CR140_Horz_Cyl_3(
	Auto:=OP140_AutoSelected , 
	Manual:=OP140_ManualSelected , 
	ErrorActive:=OP140_ErrorActive , 
	ResetPB:=OP140_HMI_Reset , 
	Sensor1:=I140_HORZ_SUP3_CYL_REVI1310_6  , 
	Sensor2:=I140_HORZ_SUP3_CYL_FWDI1310_7  , 
	ManualPB1:= , 
	ManualPB2:= , 
	AutoCmd1:= , 
	AutoCmd2:= , 
	OperationEnable:=OperationEnable , 
	SafeHome:= , 
	SafeWork:= , 
	HomingCmd1:= , 
	Pulse_1Sec:=Pulse_Block.Q1Hz , 
	BlinkingBit:= , 
	TimeOut1:=10 , 
	TimeOut2:=10 , 
	TimeOut3:=10 , 
	Solenoid1=>O140_HORZ_SUP3_CYL_REV_Q1343_0 , 
	Solenoid2=>O140_HORZ_SUP3_CYL_FWD_Q1343_1  , 
	AlarmSensor1=>berror[1331] , 
	AlarmSensor2=>berror[1332] , 
	AlarmSolenoid1=>berror[1333] , 
	AlarmSolenoid2=>berror[1334] , 
	AllSignal=>berror[1335] , 
	AlarmPresent=> , 
	Position1=> , 
	Position2=> , 
	HomeSensorBlink=> , 
	WorkSensorBlink=> , 
	Status:=OP140_GVL.CR140_Horz_Cyl_1_Status );
	
	
	//Vertical Cylinder 1
OP140_Gvl.CR140_Vert_Cyl_1_Status:=0;
// Safe Home
IF (SR140_HMI_Vert_Servo_MC1.actualPosition<=50) THEN 
	CR140_Vert_Cyl_1.SafeHome:= TRUE;
	ELSE
		CR140_Vert_Cyl_1.SafeHome:= FALSE;
	END_IF
	//Safe Work
IF(TRUE) THEN 
CR140_Vert_Cyl_1.SafeWork:=TRUE;
ELSE
	CR140_Vert_Cyl_1.SafeWork:=FALSE;
	END_IF
//Manual PB 1
IF(OP140_HMI_Vert_Cyl1_Home_PB) THEN
	CR140_Vert_Cyl_1.ManualPB1:=TRUE;
	ELSE
		CR140_Vert_Cyl_1.ManualPB1:=FALSE;
	END_IF
//Manual PB2 
IF(OP140_HMI_Vert_Cyl1_Work_PB) THEN
	CR140_Vert_Cyl_1.ManualPB2:=TRUE;
	ELSE
		CR140_Vert_Cyl_1.ManualPB2:=FALSE;
	END_IF	

	

CR140_Vert_Cyl_1(
	Auto:=OP140_AutoSelected , 
	Manual:=OP140_ManualSelected , 
	ErrorActive:=OP140_ErrorActive , 
	ResetPB:=OP140_HMI_Reset , 
	Sensor1:=I140_VERT_SUP1_CYL_REVI1301_2  , 
	Sensor2:=I140_VERT_SUP1_CYL_FWDI1301_3  , 
	ManualPB1:= , 
	ManualPB2:= , 
	AutoCmd1:= , 
	AutoCmd2:= , 
	OperationEnable:=OperationEnable , 
	SafeHome:= , 
	SafeWork:= , 
	HomingCmd1:= , 
	Pulse_1Sec:=Pulse_Block.Q1Hz  , 
	BlinkingBit:= , 
	TimeOut1:=10 , 
	TimeOut2:=10 , 
	TimeOut3:=10 , 
	Solenoid1=>O140_VERT_SUP1_CYL_REV_Q1341_2  , 
	Solenoid2=>O140_VERT_SUP1_CYL_FWD_Q1341_3 , 
	AlarmSensor1=> berror[1306], 
	AlarmSensor2=>berror[1307] , 
	AlarmSolenoid1=>berror[1308] , 
	AlarmSolenoid2=>berror[1309] , 
	AllSignal=>berror[1310],
	AlarmPresent=> , 
	Position1=> , 
	Position2=> , 
	HomeSensorBlink=> , 
	WorkSensorBlink=> , 
	Status:=OP140_Gvl.CR140_Vert_Cyl_1_Status );
	
		//Vertical Cylinder 2
CR140_Vert_Cyl_2_Status:=0;
// Safe Home
IF (SR140_HMI_Vert_Servo_MC2.actualPosition<=50) THEN 
	CR140_Vert_Cyl_2.SafeHome:= TRUE;
	ELSE
		CR140_Vert_Cyl_2.SafeHome:= FALSE;
	END_IF
	//Safe Work
IF(TRUE) THEN 
CR140_Vert_Cyl_2.SafeWork:=TRUE;
ELSE
	CR140_Vert_Cyl_2.SafeWork:=FALSE;
	END_IF
//Manual PB 1
IF(OP140_HMI_Vert_Cyl2_Home_PB) THEN
	CR140_Vert_Cyl_2.ManualPB1:=TRUE;
	ELSE
		CR140_Vert_Cyl_2.ManualPB1:=FALSE;
	END_IF
//Manual PB2 
IF(OP140_HMI_Vert_Cyl2_Work_PB) THEN
	CR140_Vert_Cyl_2.ManualPB2:=TRUE;
	ELSE
		CR140_Vert_Cyl_2.ManualPB2:=FALSE;
	END_IF	

	

CR140_Vert_Cyl_2(
	Auto:=OP140_AutoSelected , 
	Manual:=OP140_ManualSelected , 
	ErrorActive:=OP140_ErrorActive , 
	ResetPB:=OP140_HMI_Reset , 
	Sensor1:=I140_VERT_SUP2_CYL_REVI1310_2 , 
	Sensor2:=I140_VERT_SUP2_CYL_FWDI1310_3 , 
	ManualPB1:= , 
	ManualPB2:= , 
	AutoCmd1:= , 
	AutoCmd2:= , 
	OperationEnable:=OperationEnable , 
	SafeHome:= , 
	SafeWork:= , 
	HomingCmd1:= , 
	Pulse_1Sec:=Pulse_Block.Q1Hz , 
	BlinkingBit:= , 
	TimeOut1:=10 , 
	TimeOut2:=10 , 
	TimeOut3:=10 , 
	Solenoid1=>O140_VERT_SUP2_CYL_REV_Q1342_2 , 
	Solenoid2=>O140_VERT_SUP2_CYL_FWD_Q1342_3  , 
	AlarmSensor1=>berror[1321] , 
	AlarmSensor2=>berror[1322] , 
	AlarmSolenoid1=>berror[1323] , 
	AlarmSolenoid2=>berror[1324] , 
	AllSignal=>berror[1325] , 
	AlarmPresent=> , 
	Position1=> , 
	Position2=> , 
	HomeSensorBlink=> , 
	WorkSensorBlink=> , 
	Status:=CR140_Vert_Cyl_2_Status );
	
		//Vertical Cylinder 3
CR140_Vert_Cyl_3_Status:=0;
// Safe Home
IF (SR140_HMI_Vert_Servo_MC3.actualPosition<=50) THEN 
	CR140_Vert_Cyl_3.SafeHome:= TRUE;
	ELSE
		CR140_Vert_Cyl_3.SafeHome:= FALSE;
	END_IF
	//Safe Work
IF(TRUE) THEN 
   CR140_Vert_Cyl_3.SafeWork:=TRUE;
ELSE
	CR140_Vert_Cyl_3.SafeWork:=FALSE;
END_IF
//Manual PB 1
IF(OP140_HMI_Vert_Cyl3_Home_PB) THEN
	CR140_Vert_Cyl_3.ManualPB1:=TRUE;
	ELSE
		CR140_Vert_Cyl_3.ManualPB1:=FALSE;
	END_IF
//Manual PB2 
IF(OP140_HMI_Vert_Cyl3_Work_PB) THEN
	CR140_Vert_Cyl_3.ManualPB2:=TRUE;
	ELSE
		CR140_Vert_Cyl_3.ManualPB2:=FALSE;
	END_IF	

	

CR140_Vert_Cyl_3(
	Auto:=OP140_AutoSelected , 
	Manual:=OP140_ManualSelected , 
	ErrorActive:=OP140_ErrorActive , 
	ResetPB:=OP140_HMI_Reset , 
	Sensor1:=I140_VERT_SUP3_CYL_REVI1311_0 , 
	Sensor2:=I140_VERT_SUP3_CYL_FWDI1311_1  , 
	ManualPB1:= , 
	ManualPB2:= , 
	AutoCmd1:= , 
	AutoCmd2:= , 
	OperationEnable:= OperationEnable, 
	SafeHome:= , 
	SafeWork:= , 
	HomingCmd1:= , 
	Pulse_1Sec:=Pulse_Block.Q1Hz , 
	BlinkingBit:= , 
	TimeOut1:=10 , 
	TimeOut2:=10 , 
	TimeOut3:=10 , 
	Solenoid1=>O140_VERT_SUP3_CYL_REV_Q1343_2 , 
	Solenoid2=>O140_VERT_SUP3_CYL_FWD_Q1343_3  , 
	AlarmSensor1=>berror[1336] , 
	AlarmSensor2=>berror[1337] , 
	AlarmSolenoid1=>berror[1338] , 
	AlarmSolenoid2=>berror[1339] , 
	AllSignal=>berror[1340] , 
	AlarmPresent=> , 
	Position1=> , 
	Position2=> , 
	HomeSensorBlink=> , 
	WorkSensorBlink=> , 
	Status:=CR140_Vert_Cyl_3_Status );
	
		//Top Wipe Cylinder 
CR140_Wipe_Cyl_1_Status:=0;
// Safe Home
IF (TRUE) THEN 
	CR140_Top_Wipe_Cyl_1.SafeHome:= TRUE;
	ELSE
		CR140_Top_Wipe_Cyl_1.SafeHome:= FALSE;
	END_IF
	//Safe Work
IF(SR140_Vert_Servo_Ctrl_1.Axis_In_Home) THEN 
CR140_Top_Wipe_Cyl_1.SafeWork:=TRUE;
ELSE
	CR140_Top_Wipe_Cyl_1.SafeWork:=FALSE;
	END_IF
//Manual PB 1
IF(OP140_HMI_Wipe_Cyl1_Home_PB) THEN
	CR140_Top_Wipe_Cyl_1.ManualPB1:=TRUE;
	ELSE
		CR140_Top_Wipe_Cyl_1.ManualPB1:=FALSE;
	END_IF
//Manual PB2 
IF(OP140_HMI_Wipe_Cyl1_Work_PB) THEN
	CR140_Top_Wipe_Cyl_1.ManualPB2:=TRUE;
	ELSE
		CR140_Top_Wipe_Cyl_1.ManualPB2:=FALSE;
	END_IF	

	

CR140_Top_Wipe_Cyl_1(
	Auto:=OP140_AutoSelected , 
	Manual:=OP140_ManualSelected, 
	ErrorActive:=OP140_ErrorActive , 
	ResetPB:=OP140_HMI_Reset , 
	Sensor1:=I140_WIPE1_CYL_REVI1301_4, 
	Sensor2:=I140_WIPE1_CYL_FWDI1301_5 , 
	ManualPB1:= , 
	ManualPB2:= , 
	AutoCmd1:= , 
	AutoCmd2:= , 
	OperationEnable:=OperationEnable , 
	SafeHome:= , 
	SafeWork:= , 
	HomingCmd1:= , 
	Pulse_1Sec:=Pulse_Block.Q1Hz , 
	BlinkingBit:= , 
	TimeOut1:=10 , 
	TimeOut2:=10 , 
	TimeOut3:=10 , 
	Solenoid1=>O140_WIPE1_CYL_REV_Q1341_6 , 
	Solenoid2=>O140_WIPE1_CYL_FWD_Q1341_7  , 
	AlarmSensor1=>berror[1311] , 
	AlarmSensor2=>berror[1312] , 
	AlarmSolenoid1=>berror[1313] , 
	AlarmSolenoid2=>berror[1314] , 
	AllSignal=>berror[1315] , 
	AlarmPresent=> , 
	Position1=> , 
	Position2=> , 
	HomeSensorBlink=> , 
	WorkSensorBlink=> , 
	Status:=CR140_Wipe_Cyl_1_Status );
	
	//Top Wipe Cyl 2
	CR140_Wipe_Cyl_2_Status:=0;
// Safe Home
IF (TRUE) THEN 
	CR140_Top_Wipe_Cyl_2.SafeHome:= TRUE;
	ELSE
		CR140_Top_Wipe_Cyl_2.SafeHome:= FALSE;
	END_IF
	//Safe Work
IF(SR140_Vert_Servo_Ctrl_2.Axis_In_Home) THEN 
CR140_Top_Wipe_Cyl_2.SafeWork:=TRUE;
ELSE
	CR140_Top_Wipe_Cyl_2.SafeWork:=FALSE;
	END_IF
//Manual PB 1
IF(OP140_HMI_Wipe_Cyl2_Home_PB) THEN
	CR140_Top_Wipe_Cyl_2.ManualPB1:=TRUE;
	ELSE
		CR140_Top_Wipe_Cyl_2.ManualPB1:=FALSE;
	END_IF
//Manual PB2 
IF(OP140_HMI_Wipe_Cyl2_Work_PB) THEN
	CR140_Top_Wipe_Cyl_2.ManualPB2:=TRUE;
	ELSE
		CR140_Top_Wipe_Cyl_2.ManualPB2:=FALSE;
	END_IF	

	

CR140_Top_Wipe_Cyl_2(
	Auto:=OP140_AutoSelected , 
	Manual:=OP140_ManualSelected , 
	ErrorActive:=OP140_ErrorActive , 
	ResetPB:=OP140_HMI_Reset , 
	Sensor1:=I140_WIPE2_CYL_REVI1310_4 , 
	Sensor2:=I140_WIPE2_CYL_FWDI1310_5  , 
	ManualPB1:= , 
	ManualPB2:= , 
	AutoCmd1:= , 
	AutoCmd2:= , 
	OperationEnable:=OperationEnable , 
	SafeHome:= , 
	SafeWork:= , 
	HomingCmd1:= , 
	Pulse_1Sec:=Pulse_Block.Q1Hz , 
	BlinkingBit:= , 
	TimeOut1:=10 , 
	TimeOut2:=10 , 
	TimeOut3:=10 , 
	Solenoid1=>O140_WIPE2_CYL_REV_Q1342_6  , 
	Solenoid2=>O140_WIPE2_CYL_FWD_Q1342_7 , 
	AlarmSensor1=>berror[1326] , 
	AlarmSensor2=>berror[1327] , 
	AlarmSolenoid1=>berror[1328] , 
	AlarmSolenoid2=>berror[1329] , 
	AllSignal=>berror[1330] , 
	AlarmPresent=> , 
	Position1=> , 
	Position2=> , 
	HomeSensorBlink=> , 
	WorkSensorBlink=> , 
	Status:=CR140_Wipe_Cyl_2_Status );
	
//Wipe Cylinder 3

CR140_Wipe_Cyl_3_Status:=0;
// Safe Home
IF (TRUE) THEN 
	CR140_Top_Wipe_Cyl_3.SafeHome:= TRUE;
	ELSE
		CR140_Top_Wipe_Cyl_3.SafeHome:= FALSE;
	END_IF
	//Safe Work
IF(SR140_Vert_Servo_Ctrl_3.Axis_In_Home) THEN 
CR140_Top_Wipe_Cyl_3.SafeWork:=TRUE;
ELSE
	CR140_Top_Wipe_Cyl_3.SafeWork:=FALSE;
	END_IF
//Manual PB 1
IF(OP140_HMI_Wipe_Cyl3_Home_PB) THEN
	CR140_Top_Wipe_Cyl_3.ManualPB1:=TRUE;
	ELSE
		CR140_Top_Wipe_Cyl_3.ManualPB1:=FALSE;
	END_IF
//Manual PB2 
IF(OP140_HMI_Wipe_Cyl3_Work_PB) THEN
	CR140_Top_Wipe_Cyl_3.ManualPB2:=TRUE;
	ELSE
		CR140_Top_Wipe_Cyl_3.ManualPB2:=FALSE;
	END_IF	

	

CR140_Top_Wipe_Cyl_3(
	Auto:=OP140_AutoSelected , 
	Manual:=OP140_ManualSelected , 
	ErrorActive:=OP140_ErrorActive , 
	ResetPB:=OP140_HMI_Reset , 
	Sensor1:=I140_WIPE3_CYL_REVI1311_2 , 
	Sensor2:=I140_WIPE3_CYL_FWDI1311_3  , 
	ManualPB1:= , 
	ManualPB2:= , 
	AutoCmd1:= , 
	AutoCmd2:= , 
	OperationEnable:=OperationEnable , 
	SafeHome:= , 
	SafeWork:= , 
	HomingCmd1:= , 
	Pulse_1Sec:= Pulse_Block.Q1Hz, 
	BlinkingBit:= , 
	TimeOut1:=10 , 
	TimeOut2:=10 , 
	TimeOut3:= 10, 
	Solenoid1=>O140_WIPE3_CYL_REV_Q1343_6 , 
	Solenoid2=>O140_WIPE3_CYL_FWD_Q1343_7  , 
	AlarmSensor1=>berror[1341] , 
	AlarmSensor2=>berror[1342] , 
	AlarmSolenoid1=>berror[1343] , 
	AlarmSolenoid2=>berror[1344] , 
	AllSignal=>berror[1345] , 
	AlarmPresent=> , 
	Position1=> , 
	Position2=> , 
	HomeSensorBlink=> , 
	WorkSensorBlink=> , 
	Status:=CR140_Wipe_Cyl_3_Status );
		
	
	//Vertical Servo 1
	
	// Safe to Move
	
	IF CR140_Top_Wipe_Cyl_1.Position1	AND CR140_Horz_Cyl_1.Sensor2  AND CR140_Vert_Cyl_1.Position2 THEN //OR SR140_HMI_Vert_Servo_MC1.actualPosition <=50)	THEN
		
		OP140_Servo1_Safety:=TRUE;
		ELSE
			OP140_Servo1_Safety:=FALSE;
		END_IF

		//LH Vertical Servo 1
SR140_Vert_Servo_1(
	bAxis1_Ref_Switch:= , 
	bInit:= , 
	bErrorReset:=OP140_HMI_Reset OR Servo_Reset, 
	bEnable:= Servo_Enable, 
	bMoveVelocity:= , 
	bHalt:= , 
	bManualMode:=OP140_ManualSelected , 
	fHomePos:= , 
	fOverride:=100 , 
	fTargetPosition:=SR140_Vert_Servo_Ctrl_1.Position , 
	fTargetVelocity:=SR140_Vert_Servo_Ctrl_1.Velocity , 
	fAcc:= , 
	fDec:= ,
	Servo_High_Limit:= SR140_Vert_Servo_Max_Lim,	
	Servo_Low_Limit:=SR140_Vert_Servo_Min_Lim,	 	
	WARNING_LIMIT:=1,
	Safe_move_Conditions:=OP140_Servo1_Safety , 
	Axis:= SR140_Vert_Servo_Axis_1, 
	HME_WRITE_ADD:= 16#5016,	
	bHome:=SR140_Vert_Servo_Ctrl_1.Reference_Start, 
	bSetPosition:=SR140_Vert_Servo_Ctrl_1.BsetPos , 
	bMoveAbsolute:=SR140_Vert_Servo_Ctrl_1.ABSmove_Start , 
	bMoveRelative:=SR140_Vert_Servo_Ctrl_1.RELmove_Start , 
	bMoveTorque:=SR140_Vert_Servo_Ctrl_1.Torque_mode_Start , 
	stManualModeAxis:=SR140_HMI_Vert_Servo_MC1 , 
	bmove_home:=SR140_Vert_Servo_Ctrl_1.Axis_Home_Cmd , 
	sAxisState=>SR140_Vert_Servo_Ctrl_1.Axis_State , 
	bAxis_ready=>SR140_Vert_Servo_Ctrl_1.Axis_ready , 
	bAxisInPosition=>SR140_Vert_Servo_Ctrl_1.Axis_In_Pos , 
	bAxisError=>berror[1350] , 
	bAxisEnabled=>SR140_Vert_Servo_Ctrl_1.Axis_Enabled, 
	bAxisHomed=>SR140_Vert_Servo_Ctrl_1.Axis_reference  , 
	bSetPositionDone=> , 
	bHaltDone=> SR140_Vert_Servo_Ctrl_1.Axis_Halted, 
	bSTOPDone=> SR140_Vert_Servo_Ctrl_1.Axis_Stopped, 
	bHomeDone=> , 
	bDone=> , 
	bTorqueReached=>SR140_Vert_Servo_Ctrl_1.Trq_reached , 
	bsafe_to_move=>SR140_Vert_Servo_Ctrl_1.Safe_To_Move , 
	baxis_in_home_pos=>SR140_Vert_Servo_Ctrl_1.Axis_In_Home , 
	bABS_Pos_done=>, 
	Actual_position=> SR140_Vert_Servo_Ctrl_1.Actual_Position, 
	Actual_velocity=> SR140_Vert_Servo_Ctrl_1.Actual_Velocity, 
	Actual_Torque=>SR140_Vert_Servo_Ctrl_1.Actual_Torque );
	
	//Vertical Servo 2
	
	// Safe to Move
	
	IF CR140_Top_Wipe_Cyl_2.Position1 AND CR140_Horz_Cyl_2.Position2 AND CR140_Vert_Cyl_2.Position2 THEN //OR SR140_HMI_Vert_Servo_MC2.actualPosition <=50)	THEN
		
		OP140_Servo2_Safety:=TRUE;
		ELSE
			OP140_Servo2_Safety:=FALSE;
		END_IF

SR140_Vert_Servo_2(
	bAxis1_Ref_Switch:= , 
	bInit:= , 
	bErrorReset:=OP140_HMI_Reset OR Servo_Reset, 
	bEnable:= Servo_Enable, 
	bMoveVelocity:= , 
	bHalt:= , 
	bManualMode:=OP140_ManualSelected , 
	fHomePos:= , 
	fOverride:=100 , 
	fTargetPosition:= sr140_vert_servo_ctrl_2.Position, 
	fTargetVelocity:=sr140_vert_servo_ctrl_2.Velocity , 
	fAcc:= , 
	fDec:= ,
	Servo_High_Limit:= SR140_Vert_Servo_Max_Lim,	
	Servo_Low_Limit:=SR140_Vert_Servo_Min_Lim,	 	
	WARNING_LIMIT:=1, 
	Safe_move_Conditions:=OP140_Servo2_Safety OR temp, 
	Axis:= SR140_Vert_Servo_Axis_2, 
	HME_WRITE_ADD:= 16#5014,	
	bHome:=SR140_Vert_Servo_Ctrl_2.Reference_Start, 
	bSetPosition:=SR140_Vert_Servo_Ctrl_2.BsetPos , 
	bMoveAbsolute:=SR140_Vert_Servo_Ctrl_2.ABSmove_Start , 
	bMoveRelative:=SR140_Vert_Servo_Ctrl_2.RELmove_Start , 
	bMoveTorque:=SR140_Vert_Servo_Ctrl_2.Torque_mode_Start , 
	stManualModeAxis:=SR140_HMI_Vert_Servo_MC2 , 
	bmove_home:=SR140_Vert_Servo_Ctrl_2.Axis_Home_Cmd , 
	sAxisState=>SR140_Vert_Servo_Ctrl_2.Axis_State , 
	bAxis_ready=>SR140_Vert_Servo_Ctrl_2.Axis_ready , 
	bAxisInPosition=>SR140_Vert_Servo_Ctrl_2.Axis_In_Pos , 
	bAxisError=>berror[1351] , 
	bAxisEnabled=>SR140_Vert_Servo_Ctrl_2.Axis_Enabled, 
	bAxisHomed=>SR140_Vert_Servo_Ctrl_2.Axis_reference  , 
	bSetPositionDone=> , 
	bHaltDone=> SR140_Vert_Servo_Ctrl_2.Axis_Halted, 
	bSTOPDone=> SR140_Vert_Servo_Ctrl_2.Axis_Stopped, 
	bHomeDone=> , 
	bDone=> , 
	bTorqueReached=>SR140_Vert_Servo_Ctrl_2.Trq_reached , 
	bsafe_to_move=>SR140_Vert_Servo_Ctrl_2.Safe_To_Move , 
	baxis_in_home_pos=>SR140_Vert_Servo_Ctrl_2.Axis_In_Home , 
	bABS_Pos_done=> , 
	Actual_position=> SR140_Vert_Servo_Ctrl_2.Actual_Position, 
	Actual_velocity=> SR140_Vert_Servo_Ctrl_1.Actual_Velocity, 
	Actual_Torque=>SR140_Vert_Servo_Ctrl_1.Actual_Torque );
	
		//Vertical Servo 3
	
	// Safe to Move
	
	IF CR140_Top_Wipe_Cyl_3.Position1	AND CR140_Horz_Cyl_3.Sensor2  AND CR140_Vert_Cyl_3.Position2 THEN //OR  SR140_HMI_Vert_Servo_MC3.actualPosition <=50)	THEN
		
		OP140_Servo3_Safety:=TRUE;
		ELSE
			OP140_Servo3_Safety:=FALSE;
		END_IF

SR140_Vert_Servo_3(
	bAxis1_Ref_Switch:= , 
	bInit:= , 
	bErrorReset:=OP140_HMI_Reset OR Servo_Reset , 
	bEnable:= Servo_Enable, 
	bMoveVelocity:= , 
	bHalt:= , 
	bManualMode:= OP140_ManualSelected, 
	fHomePos:= , 
	fOverride:= 100, 
	fTargetPosition:=SR140_Vert_Servo_Ctrl_3.Position , 
	fTargetVelocity:=SR140_Vert_Servo_Ctrl_3.Velocity , 
	fAcc:= , 
	fDec:= ,
	Servo_High_Limit:= SR140_Vert_Servo_Max_Lim,	
	Servo_Low_Limit:=SR140_Vert_Servo_Min_Lim,	 	
	WARNING_LIMIT:=1, 
	Safe_move_Conditions:=OP140_Servo3_Safety  , 
	Axis:= SR140_Vert_Servo_Axis_3,
	HME_WRITE_ADD:= 16#5015, 
	bHome:=SR140_Vert_Servo_Ctrl_3.Reference_Start, 
	bSetPosition:=SR140_Vert_Servo_Ctrl_3.BsetPos , 
	bMoveAbsolute:=SR140_Vert_Servo_Ctrl_3.ABSmove_Start , 
	bMoveRelative:=SR140_Vert_Servo_Ctrl_3.RELmove_Start , 
	bMoveTorque:=SR140_Vert_Servo_Ctrl_3.Torque_mode_Start , 
	stManualModeAxis:=SR140_HMI_Vert_Servo_MC3 , 
	bmove_home:=SR140_Vert_Servo_Ctrl_3.Axis_Home_Cmd , 
	sAxisState=>SR140_Vert_Servo_Ctrl_3.Axis_State , 
	bAxis_ready=>SR140_Vert_Servo_Ctrl_3.Axis_ready , 
	bAxisInPosition=>SR140_Vert_Servo_Ctrl_3.Axis_In_Pos , 
	bAxisError=>berror[1352] , 
	bAxisEnabled=>SR140_Vert_Servo_Ctrl_3.Axis_Enabled, 
	bAxisHomed=>SR140_Vert_Servo_Ctrl_3.Axis_reference  , 
	bSetPositionDone=> , 
	bHaltDone=> SR140_Vert_Servo_Ctrl_3.Axis_Halted, 
	bSTOPDone=> SR140_Vert_Servo_Ctrl_3.Axis_Stopped, 
	bHomeDone=> , 
	bDone=> , 
	bTorqueReached=>SR140_Vert_Servo_Ctrl_3.Trq_reached , 
	bsafe_to_move=>SR140_Vert_Servo_Ctrl_3.Safe_To_Move , 
	baxis_in_home_pos=>SR140_Vert_Servo_Ctrl_3.Axis_In_Home , 
	bABS_Pos_done=> , 
	Actual_position=> SR140_Vert_Servo_Ctrl_3.Actual_Position, 
	Actual_velocity=>SR140_Vert_Servo_Ctrl_3.Actual_Velocity , 
	Actual_Torque=>SR140_Vert_Servo_Ctrl_3.Actual_Torque );

IF OP140_ManualSelected THEN
SR140_HMI_Vert_Servo_MC1.targetVelocity:=5;
SR140_HMI_Vert_Servo_MC2.targetVelocity:=5;
SR140_HMI_Vert_Servo_MC3.targetVelocity:=5;
END_IF

END_PROGRAM

// ---- POUs/Programs/OP140/Ateq_Comm_Prog.TcPOU
PROGRAM Ateq_Comm_Prog
VAR
	
	Pcom_In_All AT %I*: ARRAY[1..6] OF EL6inData22B;
	Pcom_Out_All AT %Q*: ARRAY[1..6] OF EL6outData22B;	
	sReceived_Data_All: ARRAY[1..6] OF STRING(255);
	BioMetric_Data	  : STRING(255);
	
	Ateq_1:SerialLineControl;
	Ateq_2:SerialLineControl;
	Ateq_3:SerialLineControl;
	Ateq_4:SerialLineControl;
	Ateq_5:SerialLineControl;
	Ateq_6:SerialLineControl;
	
	Ateq_data_1:ReceiveString255;
	Ateq_data_2:ReceiveString255;
	Ateq_data_3:ReceiveString255;
	Ateq_data_4:ReceiveString255;
	Ateq_data_5:ReceiveString255;
	Ateq_data_6:ReceiveString255;	
	BioMetric_data_FB :ReceiveString255;
	
	
	TxBuffer_1: COMbuffer;
	TxBuffer_2: COMbuffer;
	TxBuffer_3: COMbuffer;
	TxBuffer_4: COMbuffer;
	TxBuffer_5: COMbuffer;
	TxBuffer_6: COMbuffer;		
	
	RxBuffer_1: COMbuffer;
	RxBuffer_2: COMbuffer;
	RxBuffer_3: COMbuffer;
	RxBuffer_4: COMbuffer;
	RxBuffer_5: COMbuffer;
	RxBuffer_6: COMbuffer;	
	
	
	iError_ID_1: ComError_t;
    iError_ID_2: ComError_t;
	iError_ID_3: ComError_t;
	iError_ID_4: ComError_t;
	iError_ID_5: ComError_t;
	iError_ID_6: ComError_t;	
	
	
	bError_1: BOOL;
	bError_2: BOOL;
    bError_3: BOOL;
	bError_4: BOOL;		
	bError_5: BOOL;
	bError_6: BOOL;	
END_VAR

////////////////////////////////	

Ateq_1(
	Mode:= , 
	pComIn:=(ADR(Pcom_In_All[1])) , 
	pComOut:=(ADR(Pcom_Out_All[1])) , 
	SizeComIn:=SIZEOF(Pcom_In_All[1]) , 
	Error=> bError_1, 
	ErrorID=>iError_ID_1 , 
	TxBuffer:= TxBuffer_1, 
	RxBuffer:=RxBuffer_1 );

Ateq_data_1(
	Prefix:='', 
	Suffix:='' , 
	Timeout:= T#1S, 
	Reset:= (Pulse_Block.Q1Hz AND NOT Ateq_data_1.Busy) , 
	StringReceived=> , 
	Busy=> , 
	Error=> , 
	RxTimeout=> , 
	ReceivedString:= sReceived_Data_All[1], 
	RXbuffer:= RxBuffer_1);	

Ateq_2(
	Mode:= , 
	pComIn:=(ADR(Pcom_In_All[2])) , 
	pComOut:=(ADR(Pcom_Out_All[2])) , 
	SizeComIn:=SIZEOF(Pcom_In_All[2]) , 
	Error=> bError_2, 
	ErrorID=>iError_ID_2 , 
	TxBuffer:= TxBuffer_2, 
	RxBuffer:=RxBuffer_2 );

Ateq_data_2(
	Prefix:='', 
	Suffix:='' , 
	Timeout:= T#1S, 
	Reset:= (Pulse_Block.Q1Hz AND NOT Ateq_data_2.Busy) , 
	StringReceived=> , 
	Busy=> , 
	Error=> , 
	RxTimeout=> , 
	ReceivedString:= sReceived_Data_All[2], 
	RXbuffer:= RxBuffer_2);	
	
Ateq_3(
	Mode:= , 
	pComIn:=(ADR(Pcom_In_All[3])) , 
	pComOut:=(ADR(Pcom_Out_All[3])) , 
	SizeComIn:=SIZEOF(Pcom_In_All[3]) , 
	Error=> bError_3, 
	ErrorID=>iError_ID_3 , 
	TxBuffer:= TxBuffer_3, 
	RxBuffer:=RxBuffer_3 );

Ateq_data_3(
	Prefix:='', 
	Suffix:='' , 
	Timeout:= T#1S, 
	Reset:= (Pulse_Block.Q1Hz AND NOT Ateq_data_3.Busy) , 
	StringReceived=> , 
	Busy=> , 
	Error=> , 
	RxTimeout=> , 
	ReceivedString:= sReceived_Data_All[3], 
	RXbuffer:= RxBuffer_3);	


Ateq_4(
	Mode:= , 
	pComIn:=(ADR(Pcom_In_All[4])) , 
	pComOut:=(ADR(Pcom_Out_All[4])) , 
	SizeComIn:=SIZEOF(Pcom_In_All[4]) , 
	Error=> bError_4, 
	ErrorID=>iError_ID_4 , 
	TxBuffer:= TxBuffer_4, 
	RxBuffer:=RxBuffer_4 );

Ateq_data_4(
	Prefix:='', 
	Suffix:='' , 
	Timeout:= T#1S, 
	Reset:= (Pulse_Block.Q1Hz AND NOT Ateq_data_4.Busy) , 
	StringReceived=> , 
	Busy=> , 
	Error=> , 
	RxTimeout=> , 
	ReceivedString:= sReceived_Data_All[4], 
	RXbuffer:= RxBuffer_4);

Ateq_5(
	Mode:= , 
	pComIn:=(ADR(Pcom_In_All[5])) , 
	pComOut:=(ADR(Pcom_Out_All[5])) , 
	SizeComIn:=SIZEOF(Pcom_In_All[5]) , 
	Error=> bError_5, 
	ErrorID=>iError_ID_5 , 
	TxBuffer:= TxBuffer_5, 
	RxBuffer:=RxBuffer_5 );

Ateq_data_5(
	Prefix:='', 
	Suffix:='' , 
	Timeout:= T#1S, 
	Reset:= (Pulse_Block.Q1Hz AND NOT Ateq_data_5.Busy) , 
	StringReceived=> , 
	Busy=> , 
	Error=> , 
	RxTimeout=> , 
	ReceivedString:= sReceived_Data_All[5], 
	RXbuffer:= RxBuffer_5);	


Ateq_6(
	Mode:= , 
	pComIn:=(ADR(Pcom_In_All[6])) , 
	pComOut:=(ADR(Pcom_Out_All[6])) , 
	SizeComIn:=SIZEOF(Pcom_In_All[6]) , 
	Error=> bError_6, 
	ErrorID=>iError_ID_6 , 
	TxBuffer:= TxBuffer_6, 
	RxBuffer:=RxBuffer_6 );

Ateq_data_6(
	Prefix:='', 
	Suffix:='' , 
	Timeout:= T#1S, 
	Reset:= (Pulse_Block.Q1Hz AND NOT Ateq_data_6.Busy) , 
	StringReceived=> , 
	Busy=> , 
	Error=> , 
	RxTimeout=> , 
	ReceivedString:= sReceived_Data_All[6], 
	RXbuffer:= RxBuffer_6);		
	
	
BioMetric_data_FB(
	Prefix:='', 
	Suffix:='', 
	Timeout:= T#1S, 
	Reset:= (Pulse_Block.Q1Hz AND NOT BioMetric_data_FB.Busy) , 
	StringReceived=> , 
	Busy=> , 
	Error=> , 
	RxTimeout=> , 
	ReceivedString:= BioMetric_Data, 
	RXbuffer:= SerialComm.RxBuffer_1);

END_PROGRAM

// ---- POUs/Programs/OP140/OP140_Initialization_Seq.TcPOU
PROGRAM OP140_Initialization_Seq
VAR
	ateq_reseted :bool;
END_VAR

IF ( SR140_Vert_Servo_Ctrl_1.Axis_In_Home AND SR140_Vert_Servo_Ctrl_2.Axis_In_Home AND SR140_Vert_Servo_Ctrl_3.Axis_In_Home AND CR140_Horz_Cyl_1.Position1 
    AND  CR140_Horz_Cyl_2.Position1 AND  CR140_Horz_Cyl_3.Position1  AND  CR140_Vert_Cyl_1.Position1 AND CR140_Vert_Cyl_2.Position1 AND ateq_reseted
    AND  CR140_Vert_Cyl_3.Position1 AND CR140_Top_Wipe_Cyl_1.Position1 AND CR140_Top_Wipe_Cyl_2.Position1 AND CR140_Top_Wipe_Cyl_3.Position1 )THEN
   
    OP140_Temp_Home_Ok:=TRUE;
    OP140_HomeRunning:=FALSE;
    OP140_Homing_Seq:=0;
	
    ELSE
	OP140_Temp_Home_Ok:=FALSE;
	ateq_reseted := FALSE;
	
END_IF

CASE OP140_Homing_Seq OF
	
	   0: IF (OP140_Auto AND NOT OP140_HomeRunning AND  NOT OP140_ErrorActive AND  NOT OP140_AutoRunning AND NOT OP140_StepRunning	 AND NOT OP140_Temp_Home_Ok) THEN
		      OP140_HomeRunning:=TRUE;
		      OP140_Homing_Seq:=10;	
	      END_IF
	   
	   10:IF (OP140_HomeRunning AND OP140_HMI_Homing)THEN   /// waiting for hmi homing feedback
             OP140_ATEQ1_Auto_Start:=FALSE;
			 OP140_ATEQ2_Auto_Start:=FALSE;
			 OP140_ATEQ3_Auto_Start:=FALSE;
			 OP140_ATEQ4_Auto_Start:=FALSE;
			 OP140_ATEQ5_Auto_Start:=FALSE;
			 OP140_ATEQ6_Auto_Start:=FALSE;
			 OP140_ATEQ_Reset :=TRUE;
			 OP140_Homing_Seq:=20;
		  END_IF 
			
	  20:	CR140_Top_Wipe_Cyl_1.HomingCmd1:= TRUE; 
			CR140_Top_Wipe_Cyl_2.HomingCmd1:= TRUE; 
			CR140_Top_Wipe_Cyl_3.HomingCmd1:= TRUE; 
			
			IF CR140_Top_Wipe_Cyl_1.position1 AND CR140_Top_Wipe_Cyl_2.Position1 AND  CR140_Top_Wipe_Cyl_3.Position1=TRUE THEN
			   CR140_Top_Wipe_Cyl_1.HomingCmd1:= FALSE;
			   CR140_Top_Wipe_Cyl_2.HomingCmd1:= FALSE;
			   CR140_Top_Wipe_Cyl_3.HomingCmd1:= FALSE;
			   OP140_Homing_Seq:=30;
			END_IF
			
	 30:  SR140_Vert_Servo_Ctrl_1.Position:=0.0;
		  SR140_Vert_Servo_Ctrl_1.Velocity:=50;
		  SR140_Vert_Servo_Ctrl_2.Position:=0.0;
		  SR140_Vert_Servo_Ctrl_2.Velocity:=50;
		  SR140_Vert_Servo_Ctrl_3.Position:=0.0;
		  SR140_Vert_Servo_Ctrl_3.Velocity:=50;
		  SR140_Vert_Servo_Ctrl_1.Axis_Home_Cmd:=TRUE;
		  SR140_Vert_Servo_Ctrl_2.Axis_Home_Cmd:=TRUE;
		  SR140_Vert_Servo_Ctrl_3.Axis_Home_Cmd:=TRUE; 
		  
		  IF (SR140_Vert_Servo_Ctrl_1.Axis_In_Home AND SR140_Vert_Servo_Ctrl_2.Axis_In_Home AND SR140_Vert_Servo_Ctrl_3.Axis_In_Home)=TRUE THEN
			 SR140_Vert_Servo_Ctrl_1.Axis_Home_Cmd:=FALSE;
			 SR140_Vert_Servo_Ctrl_2.Axis_Home_Cmd:=FALSE;
			 SR140_Vert_Servo_Ctrl_3.Axis_Home_Cmd:=FALSE;
			 OP140_Homing_Seq:=40;
		END_IF	
	
    40:	CR140_Vert_Cyl_1.HomingCmd1:= TRUE;	
		CR140_Vert_Cyl_2.HomingCmd1:= TRUE;	
		CR140_Vert_Cyl_3.HomingCmd1:= TRUE;	
		IF CR140_Vert_Cyl_1.Position1 AND CR140_Vert_Cyl_2.Position1 AND  CR140_Vert_Cyl_3.Position1=TRUE THEN
		   CR140_Vert_Cyl_1.HomingCmd1:= FALSE;
		   CR140_Vert_Cyl_2.HomingCmd1:= FALSE;
		   CR140_Vert_Cyl_3.HomingCmd1:= FALSE;
           OP140_Homing_Seq:=50;
		END_IF
		
	50:	CR140_Horz_Cyl_1.HomingCmd1:= TRUE;
		CR140_Horz_Cyl_2.HomingCmd1:= TRUE;
		CR140_Horz_Cyl_3.HomingCmd1:= TRUE;
		IF CR140_Horz_Cyl_1.Position1 AND  CR140_Horz_Cyl_2.Position1 AND CR140_Horz_Cyl_3.Position1 THEN
		   CR140_Horz_Cyl_1.HomingCmd1:= FALSE;
		   CR140_Horz_Cyl_2.HomingCmd1:= FALSE;
		   CR140_Horz_Cyl_3.HomingCmd1:= FALSE;
		   OP140_Homing_Seq:=60;
	    END_IF
	
    60:  OP140_ATEQ_Reset :=FALSE;
	     IF NOT  OP140_ATEQ_Reset  THEN
		    OP140_HomeRunning:=FALSE;
			OP140_ATEQ1_Auto_Start:=TRUE;
			OP140_ATEQ2_Auto_Start:=TRUE;
			OP140_ATEQ3_Auto_Start:=TRUE;
			OP140_ATEQ4_Auto_Start:=TRUE;
			OP140_ATEQ5_Auto_Start:=TRUE;
			OP140_ATEQ6_Auto_Start:=TRUE;
			ateq_reseted := TRUE;
			IF ateq_reseted THEN
			   OP140_ATEQ1_Auto_Start:=FALSE;
			   OP140_ATEQ2_Auto_Start:=FALSE;
			   OP140_ATEQ3_Auto_Start:=FALSE;
			   OP140_ATEQ4_Auto_Start:=FALSE;
			   OP140_ATEQ5_Auto_Start:=FALSE;
			   OP140_ATEQ6_Auto_Start:=FALSE;
               OP140_Homing_Seq:=0;
			END_IF
		 END_IF	
			
END_CASE		

IF NOT OP140_HomeRunning THEN
	
	CR140_Horz_Cyl_1.HomingCmd1:= FALSE;
	CR140_Horz_Cyl_2.HomingCmd1:= FALSE;
	CR140_Horz_Cyl_3.HomingCmd1:= FALSE;
	CR140_Vert_Cyl_1.HomingCmd1:= FALSE;
	CR140_Vert_Cyl_2.HomingCmd1:= FALSE;
	CR140_Vert_Cyl_3.HomingCmd1:= FALSE;
	CR140_Top_Wipe_Cyl_1.HomingCmd1:= FALSE;
	CR140_Top_Wipe_Cyl_2.HomingCmd1:= FALSE;
	CR140_Top_Wipe_Cyl_3.HomingCmd1:= FALSE;
	
END_IF
		
		
			
			
			
    (*       IF ( CR140_Top_Wipe_Cyl_1.Position1 AND CR140_Top_Wipe_Cyl_2.Position1 AND  CR140_Top_Wipe_Cyl_3.Position1=TRUE ) THEN
			    OP140_Homing_Seq:=20;
			    ELSE
				CR140_Top_Wipe_Cyl_1.HomingCmd1:= TRUE;
				CR140_Top_Wipe_Cyl_2.HomingCmd1:= TRUE;
				CR140_Top_Wipe_Cyl_3.HomingCmd1:= TRUE;
				
				IF   CR140_Top_Wipe_Cyl_1.position1 AND CR140_Top_Wipe_Cyl_2.Position1 AND  CR140_Top_Wipe_Cyl_3.Position1=TRUE THEN
				     CR140_Top_Wipe_Cyl_1.HomingCmd1:= FALSE;
				     CR140_Top_Wipe_Cyl_2.HomingCmd1:= FALSE;
				     CR140_Top_Wipe_Cyl_3.HomingCmd1:= FALSE;
				     OP140_Homing_Seq:=30;
				END_IF
			END_IF
		END_IF
		
	20:IF (OP140_HomeRunning AND OP140_HMI_Homing)THEN 
        IF (SR140_Vert_Servo_Ctrl_1.Axis_In_Home AND SR140_Vert_Servo_Ctrl_2.Axis_In_Home AND SR140_Vert_Servo_Ctrl_3.Axis_In_Home)=TRUE THEN
			OP140_Homing_Seq:=30;
			ELSE
				SR140_Vert_Servo_Ctrl_1.Position:=0.0;
				SR140_Vert_Servo_Ctrl_1.Velocity:=50;
				SR140_Vert_Servo_Ctrl_2.Position:=0.0;
				SR140_Vert_Servo_Ctrl_2.Velocity:=50;
				SR140_Vert_Servo_Ctrl_3.Position:=0.0;
				SR140_Vert_Servo_Ctrl_3.Velocity:=50;
				SR140_Vert_Servo_Ctrl_1.Axis_Home_Cmd:=TRUE;
				SR140_Vert_Servo_Ctrl_2.Axis_Home_Cmd:=TRUE;
				SR140_Vert_Servo_Ctrl_3.Axis_Home_Cmd:=TRUE;
				
				
				IF (SR140_Vert_Servo_Ctrl_1.Axis_In_Home AND SR140_Vert_Servo_Ctrl_2.Axis_In_Home AND SR140_Vert_Servo_Ctrl_3.Axis_In_Home)=TRUE THEN
				
					SR140_Vert_Servo_Ctrl_1.Axis_Home_Cmd:=FALSE;
				SR140_Vert_Servo_Ctrl_2.Axis_Home_Cmd:=FALSE;
				SR140_Vert_Servo_Ctrl_3.Axis_Home_Cmd:=FALSE;
				OP140_Homing_Seq:=30;
				END_IF
				
				END_IF
				END_IF
	30:IF (OP140_HomeRunning AND OP140_HMI_Homing)THEN 
        IF ( CR140_Vert_Cyl_1.Position1 AND CR140_Vert_Cyl_2.Position1 AND  CR140_Vert_Cyl_3.Position1=TRUE ) THEN
			OP140_Homing_Seq:=40;
			ELSE
	
				CR140_Vert_Cyl_1.HomingCmd1:= TRUE;
				CR140_Vert_Cyl_2.HomingCmd1:= TRUE;
				CR140_Vert_Cyl_3.HomingCmd1:= TRUE;
				
				IF   CR140_Vert_Cyl_1.Position1 AND CR140_Vert_Cyl_2.Position1 AND  CR140_Vert_Cyl_3.Position1=TRUE THEn
				    CR140_Vert_Cyl_1.HomingCmd1:= FALSE;
				    CR140_Vert_Cyl_2.HomingCmd1:= FALSE;
				    CR140_Vert_Cyl_3.HomingCmd1:= FALSE;
				    OP140_Homing_Seq:=40;
			   END_IF
				
				END_IF
				END_IF
		40:IF (OP140_HomeRunning AND OP140_HMI_Homing)THEN 
              IF ( CR140_Horz_Cyl_1.Position1 AND CR140_Horz_Cyl_2.Position1 AND  CR140_Horz_Cyl_3.Position1=TRUE ) THEN
			     OP140_Homing_Seq:=40;
			  ELSE
	             CR140_Horz_Cyl_1.HomingCmd1:= TRUE;
			     CR140_Horz_Cyl_2.HomingCmd1:= TRUE;
			     CR140_Horz_Cyl_3.HomingCmd1:= TRUE;
			  IF CR140_Horz_Cyl_1.Position1 AND  CR140_Horz_Cyl_2.Position1 AND CR140_Horz_Cyl_3.Position1 THEN
				 CR140_Horz_Cyl_1.HomingCmd1:= FALSE;
				 CR140_Horz_Cyl_2.HomingCmd1:= FALSE;
			     CR140_Horz_Cyl_3.HomingCmd1:= FALSE;
			     OP140_Homing_Seq:=50;
			  END_IF
				
			END_IF
		END_IF
			
  50:  OP140_ATEQ_Reset :=FALSE;
     IF NOT  OP140_ATEQ_Reset  THEN
	   OP140_HomeRunning:=FALSE;
	   OP140_Homing_Seq:=0;
	   END_IF*)

END_PROGRAM

// ---- POUs/Programs/OP140/op140_tool_change.TcPOU
PROGRAM op140_tool_change
VAR
	op140_1_tool_change : tool_changeover;
	op140_2_tool_change : tool_changeover; 
	op140_3_tool_change : tool_changeover;
	fb_reset_1       :BOOL;
	fb_reset_2       :BOOL;
	fb_reset_3       :BOOL;
	
	
	tool_6_fb: BOOL;
	tool_8_fb: BOOL;
	
	// VERTICAL 1
	OP140_V1_TOL_UNLOD_STRT					: BOOL;
	OP140_V1_TOL_LOAD_STRT					: BOOL;
	OP140_V1_TOL_DISENGAGE					: BOOL;
	OP140_V1_TOL_ENGAGE						: BOOL;
	op140_t1_manual_lock                    : BOOL;
	op140_t1_manual_unlock                  : BOOL;
	OP140_V1_UNLD_STUS                      : STRING;
	OP140_V1_LOAD_STUS                      : STRING;
	
	// VERTICAL 2
	
	OP140_V2_TOL_UNLOD_STRT					: BOOL;
	OP140_V2_TOL_LOAD_STRT					: BOOL;
	OP140_V2_TOL_DISENGAGE					: BOOL;
	OP140_V2_TOL_ENGAGE						: BOOL;
	op140_t2_manual_lock                    : BOOL;
	op140_t2_manual_unlock                  : BOOL;
	OP140_V2_UNLD_STUS                      : STRING;
	OP140_V2_LOAD_STUS                      : STRING;
	
	// VERTICAL 3
	
	OP140_V3_TOL_UNLOD_STRT					: BOOL;
	OP140_V3_TOL_LOAD_STRT					: BOOL;
	OP140_V3_TOL_DISENGAGE					: BOOL;
	OP140_V3_TOL_ENGAGE						: BOOL;
	op140_t3_manual_lock                    : BOOL;
	op140_t3_manual_unlock                  : BOOL;
	OP140_V3_UNLD_STUS                      : STRING;
	OP140_V3_LOAD_STUS                      : STRING;
	
	
END_VAR

VAR PERSISTENT
	
	OP140_V1_TOL_WRK_POS					: LREAL;
	OP140_V1_TOL_HME_POS					: LREAL;
	op140_v1_TOL_VELOCITY					: LREAL;
	OP140_V1_TOL_CHNGE_CMPLE				: BOOL;
	OP140_V1_TOL_LOAD_COMPLE                : BOOL;
	OP140_V1_TOL_UNLOAD_COMPLE              : BOOL;
	
	OP140_V2_TOL_WRK_POS					: LREAL;
	OP140_V2_TOL_HME_POS					: LREAL;
	op140_V2_T0L_VELOCITY					: LREAL;
	OP140_V2_TOL_CHNGE_CMPLE				: BOOL;
	OP140_V2_TOL_LOAD_COMPLE                : BOOL;
	OP140_V2_TOL_UNLOAD_COMPLE              : BOOL;
	
	
	OP140_V3_TOL_WRK_POS					: LREAL;
	OP140_V3_TOL_HME_POS					: LREAL;
	op140_v3_TOL_VELOCITY					: LREAL;
	OP140_V3_TOL_CHNGE_CMPLE				: BOOL;
	OP140_V3_TOL_LOAD_COMPLE                : BOOL;
	OP140_V3_TOL_UNLOAD_COMPLE              : BOOL;
	
END_VAR

IF OP140_TOOL_CHANGE_MODE_SELECTED THEN

op140_1_tool_change(
	actual_pos:= SR140_Vert_Servo_Ctrl_1.Actual_position , 
	actual_vel:=SR140_Vert_Servo_Ctrl_1.Actual_velocity , 
	target_work_pos:= OP140_V1_TOL_WRK_POS, 
	target_home_pos:= OP140_V1_TOL_HME_POS, 
	target_vel_from_hmi:= op140_v1_TOL_VELOCITY, 
	station_number:= , 
	mover_number:= , 
	no_of_mover_present:= , 
	model_selected:= model_selected, 
	tool_unloading_start:=OP140_V1_TOL_UNLOD_STRT , 
	tool_loading_start:=OP140_V1_TOL_LOAD_STRT , 
	error_active:=OP140_ErrorActive , 
	station_in_auto:= OP140_Auto, 
	station_in_home:=  OP140_Temp_Home_Ok, 
	absoulte_move_done:= SR140_Vert_Servo_Ctrl_1.Axis_In_Pos, 
	tool_6_3_present:= tool_6_fb, 
	tool_7_89_present:= tool_8_fb, 
	fb_reset:=fb_reset_1,
	SERVO_TOL_CHECK_OFFSET_POS := 18, 
	tool_changer_over_complete=> OP140_V1_TOL_CHNGE_CMPLE,
	tool_disengage=> OP140_V1_TOL_DISENGAGE, 
	tool_engagae=> OP140_V1_TOL_ENGAGE, 
	tool_loading_complete=> OP140_V1_TOL_LOAD_COMPLE, 
	tool_unloading_complete=> OP140_V1_TOL_UNLOAD_COMPLE, 
	servo_move_abs=>SR140_Vert_Servo_Ctrl_1.ABSmove_Start, 
	unloading_status=>OP140_V1_UNLD_STUS , 
	loading_status=>OP140_V1_LOAD_STUS , 
	target_pos_to_servo=>SR140_Vert_Servo_Ctrl_1.Position , 
	target_vel_to_servo=> SR140_Vert_Servo_Ctrl_1.Velocity,
tool_loading_failed := );
	
	op140_2_tool_change(
	actual_pos:= SR140_Vert_Servo_Ctrl_2.Actual_position , 
	actual_vel:=SR140_Vert_Servo_Ctrl_2.Actual_velocity , 
	target_work_pos:= OP140_V2_TOL_WRK_POS, 
	target_home_pos:= OP140_V2_TOL_HME_POS, 
	target_vel_from_hmi:= op140_V2_T0L_VELOCITY, 
	station_number:= , 
	mover_number:= , 
	no_of_mover_present:= , 
	model_selected:= model_selected, 
	tool_unloading_start:=OP140_V2_TOL_UNLOD_STRT , 
	tool_loading_start:=OP140_V2_TOL_LOAD_STRT , 
	error_active:=OP140_ErrorActive , 
	station_in_auto:= OP140_Auto, 
	station_in_home:=  OP140_Temp_Home_Ok, 
	absoulte_move_done:= SR140_Vert_Servo_Ctrl_2.Axis_In_Pos, 
	tool_6_3_present:= tool_6_fb, 
	tool_7_89_present:= tool_8_fb, 
	fb_reset:=fb_reset_1,
	SERVO_TOL_CHECK_OFFSET_POS := 18, 
	tool_changer_over_complete=> OP140_V2_TOL_CHNGE_CMPLE,
	tool_disengage=> OP140_V2_TOL_DISENGAGE, 
	tool_engagae=> OP140_V2_TOL_ENGAGE, 
	tool_loading_complete=> OP140_V2_TOL_LOAD_COMPLE, 
	tool_unloading_complete=> OP140_V2_TOL_UNLOAD_COMPLE, 
	servo_move_abs=>SR140_Vert_Servo_Ctrl_2.ABSmove_Start, 
	unloading_status=>OP140_V2_UNLD_STUS , 
	loading_status=>OP140_V2_LOAD_STUS , 
	target_pos_to_servo=>SR140_Vert_Servo_Ctrl_2.Position , 
	target_vel_to_servo=> SR140_Vert_Servo_Ctrl_2.Velocity,
tool_loading_failed := );
	
	op140_3_tool_change(
	actual_pos:= SR140_Vert_Servo_Ctrl_3.Actual_position , 
	actual_vel:=SR140_Vert_Servo_Ctrl_3.Actual_velocity , 
	target_work_pos:= OP140_V3_TOL_WRK_POS, 
	target_home_pos:= OP140_V3_TOL_HME_POS, 
	target_vel_from_hmi:= op140_v3_TOL_VELOCITY, 
	station_number:= , 
	mover_number:= , 
	no_of_mover_present:= , 
	model_selected:= model_selected, 
	tool_unloading_start:=OP140_V3_TOL_UNLOD_STRT , 
	tool_loading_start:=OP140_V3_TOL_LOAD_STRT , 
	error_active:=OP140_ErrorActive , 
	station_in_auto:= OP140_Auto, 
	station_in_home:=  OP140_Temp_Home_Ok, 
	absoulte_move_done:= SR140_Vert_Servo_Ctrl_3.Axis_In_Pos, 
	tool_6_3_present:= tool_6_fb, 
	tool_7_89_present:= tool_8_fb, 
	fb_reset:=fb_reset_1,
	SERVO_TOL_CHECK_OFFSET_POS := 18, 
	tool_changer_over_complete=> OP140_V3_TOL_CHNGE_CMPLE,
	tool_disengage=> OP140_V3_TOL_DISENGAGE, 
	tool_engagae=> OP140_V3_TOL_ENGAGE, 
	tool_loading_complete=> OP140_V3_TOL_LOAD_COMPLE, 
	tool_unloading_complete=> OP140_V3_TOL_UNLOAD_COMPLE, 
	servo_move_abs=>SR140_Vert_Servo_Ctrl_3.ABSmove_Start, 
	unloading_status=>OP140_V3_UNLD_STUS , 
	loading_status=>OP140_V3_LOAD_STUS , 
	target_pos_to_servo=>SR140_Vert_Servo_Ctrl_3.Position , 
	target_vel_to_servo=> SR140_Vert_Servo_Ctrl_3.Velocity,
tool_loading_failed := );
	
	END_IF 

//// op 140 tool 1 outputs/////

	
IF op140_t1_manual_lock OR OP140_V1_TOL_ENGAGE THEN
	O140_TOOL1_CHO_LOCK_Q1341_5:=TRUE;
	O140_TOOL1_CHO_UNLOCK_Q1341_4 :=FALSE;
ELSIF op140_t1_manual_unlock OR OP140_V1_TOL_DISENGAGE THEN
	O140_TOOL1_CHO_UNLOCK_Q1341_4 :=TRUE;
	O140_TOOL1_CHO_LOCK_Q1341_5:=FALSE;
END_IF
   

//// op 140 tool 2 outputs///// 	

IF op140_t2_manual_lock OR OP140_V2_TOL_ENGAGE THEN
	O140_TOOL2_CHO_LOCK_Q1342_5:=TRUE;
	O140_TOOL2_CHO_UNLOCK_Q1342_4 :=FALSE;
ELSIF op140_t2_manual_unlock OR OP140_V2_TOL_DISENGAGE THEN
	O140_TOOL2_CHO_UNLOCK_Q1342_4 :=TRUE;
	O140_TOOL2_CHO_LOCK_Q1342_5   :=FALSE;
END_IF

//// op 140 tool 3 outputs/////

IF op140_t3_manual_lock OR OP140_V3_TOL_ENGAGE THEN
	O140_TOOL3_CHO_LOCK_Q1343_5   :=TRUE;
	O140_TOOL3_CHO_UNLOCK_Q1343_4 :=FALSE;
ELSIF op140_t3_manual_unlock OR OP140_V3_TOL_DISENGAGE THEN
	O140_TOOL3_CHO_UNLOCK_Q1343_4 :=TRUE;
	O140_TOOL3_CHO_LOCK_Q1343_5   :=FALSE;
END_IF

END_PROGRAM

// ---- POUs/Programs/OP140/op140_ateq_fb.TcPOU
PROGRAM op140_ateq_fb
VAR
	 OP140_ATEQ1_Manual_Start:BOOL;
	 OP140_ATEQ2_Manual_Start:BOOL;
	 OP140_ATEQ3_Manual_Start:BOOL;
	 OP140_ATEQ4_Manual_Start:BOOL;
	 OP140_ATEQ5_Manual_Start:BOOL;
	 OP140_ATEQ6_Manual_Start:BOOL;
	 OP140_ATEQ1_Manual_Prog_No:INT;
	 OP140_ATEQ2_Manual_Prog_No:INT;
	 OP140_ATEQ3_Manual_Prog_No:INT;
	 OP140_ATEQ4_Manual_Prog_No:INT;
	 OP140_ATEQ5_Manual_Prog_No:INT;
	 OP140_ATEQ6_Manual_Prog_No:INT;
	 OP140_ATEQ1_Reset:BOOL;
	 OP140_ATEQ2_Reset:BOOL;
	 OP140_ATEQ3_Reset:BOOL;
	 OP140_ATEQ4_Reset:BOOL;
	 OP140_ATEQ5_Reset:BOOL;
	 OP140_ATEQ6_Reset:BOOL;
	 OP140_ATEQ1_FB:ATEQ_LEAK;
	 OP140_ATEQ2_FB:ATEQ_LEAK;
	 OP140_ATEQ3_FB:ATEQ_LEAK;
	 OP140_ATEQ4_FB:ATEQ_LEAK;
	 OP140_ATEQ5_FB:ATEQ_LEAK;
	 OP140_ATEQ6_FB:ATEQ_LEAK;
END_VAR

//HMI Sel ATEQ
CASE OP140_ATEQ_SEL_NO of
	1:
			 OP140_ATEQ1_Manual_Start:=OP140_ATEQ_Start;
			  OP140_ATEQ1_Reset:=OP140_ATEQ_Reset;
			  OP140_ATEQ1_Manual_Prog_No:=OP140_ATEQ_Prog_No;
	2:
			 OP140_ATEQ2_Manual_Start:=OP140_ATEQ_Start;
			  OP140_ATEQ2_Reset:=OP140_ATEQ_Reset;
			  OP140_ATEQ2_Manual_Prog_No:=OP140_ATEQ_Prog_No;
			  
	3:       
			 OP140_ATEQ3_Manual_Start:=OP140_ATEQ_Start;
			  OP140_ATEQ3_Reset:=OP140_ATEQ_Reset;
			  OP140_ATEQ3_Manual_Prog_No:=OP140_ATEQ_Prog_No;
			  
	4:
	
				 OP140_ATEQ4_Manual_Start:=OP140_ATEQ_Start;
			  OP140_ATEQ4_Reset:=OP140_ATEQ_Reset;
			  OP140_ATEQ4_Manual_Prog_No:=OP140_ATEQ_Prog_No;
			  
	5:			
				 OP140_ATEQ5_Manual_Start:=OP140_ATEQ_Start;
			  OP140_ATEQ5_Reset:=OP140_ATEQ_Reset;
			  OP140_ATEQ5_Manual_Prog_No:=OP140_ATEQ_Prog_No;
			  
	6:
	
				OP140_ATEQ6_Manual_Start:=OP140_ATEQ_Start;
			  OP140_ATEQ6_Reset:=OP140_ATEQ_Reset;
			  OP140_ATEQ6_Manual_Prog_No:=OP140_ATEQ_Prog_No;
	
END_CASE
IF OP140_AutoSelected THEN
   OP140_ATEQ_Start:=FALSE	;
   OP140_ATEQ1_Manual_Start:=FALSE;
   OP140_ATEQ2_Manual_Start:=FALSE;
   OP140_ATEQ3_Manual_Start:=FALSE;
   OP140_ATEQ4_Manual_Start:=FALSE;
   OP140_ATEQ5_Manual_Start:=FALSE;
   OP140_ATEQ6_Manual_Start:=FALSE;
END_IF

//ATEQ Manual Actuation
 OP140_ATEQ1_FB(
	AutoSelected:=OP140_AutoSelected , 
	ManualSelected:=OP140_ManualSelected  , 
	Manual_Start:= OP140_ATEQ1_Manual_Start , 
	Auto_Start:=OP140_ATEQ1_Auto_Start, 
	Erroractive:=OP140_ErrorActive , 
	Start:= , 
	Reset:=OP140_ATEQ_Reset  , 
	Manual_Prog_No:=  OP140_ATEQ1_Manual_Prog_No , 
	Auto_Prog_No:=OP140_ATEQ1_Auto_Prog_No_out , 
	Testpass:= I140_LK_TST_1_PASI703_3, 
	Testfail:=I140_LK_TST_1_FLI703_4 , 
	Reffail:=I140_LK_TST_1_REF_PRT_FLI703_5 , 
	Alarm:=I140_LK_TST_1_WARNGI703_6 , 
	Endofcycle:=I140_LK_TST_1_END_CYCI703_7,
	StartRSTDly:= , 
	StartOP=>O140_LK_TST1_STRT_Q700_1 , 
	ResetOP=>O140_LK_TST1_RST_Q700_0 , 
	
	Receive_String := Ateq_Comm_Prog.sReceived_Data_All[1] ,
	result_Ateq=> OP140_ATEQ1_Result,
	Prg_num=> OP140_ATEQ1_Prgrm_Num,	
    status=> OP140_ATEQ1_Status,
	Error1=> , 
	Error2=> , 
	Error3=> , 
	ProgSel1=>O140_LK_TST1_SEL1_Q700_2 , 
	ProgSel2=>O140_LK_TST1_SEL2_Q700_3 , 
	ProgSel3=> O140_LK_TST1_SEL3_Q700_4, 
	ProgSel4=> O140_LK_TST1_SEL4_Q700_5, 
	ProgSel5=>O140_LK_TST1_SEL5_Q700_6 , 
	ProgSel6=> O140_LK_TST1_SEL6_Q700_7, 
	ProgSel7=>O140_LK_TST1_SEL7_Q701_0 , 
	ProgSel8=>,
	Result_Completed:=OP140_ATEQ1_ResultCompleted ,
    ResultOK  :=OP140_ATEQ1_ResultOK , 
	ResultNOK := OP140_ATEQ1_ResultNOK );

//ATEQ 2

OP140_ATEQ2_FB(
	AutoSelected:=OP140_AutoSelected , 
	ManualSelected:=OP140_ManualSelected  , 
	Manual_Start:= OP140_ATEQ2_Manual_Start , 
	Auto_Start:=  OP140_ATEQ2_Auto_Start, 
	Erroractive:=OP140_ErrorActive , 
	Start:= , 
	Reset:=OP140_ATEQ_Reset  , 
	Manual_Prog_No:=  OP140_ATEQ2_Manual_Prog_No , 
	Auto_Prog_No:=OP140_ATEQ2_Auto_Prog_No_out , 
	Testpass:= I140_LK_TST_2_PASI704_1, 
	Testfail:=I140_LK_TST_2_FLI704_2 , 
	Reffail:=I140_LK_TST_2_REF_PRT_FLI704_3 , 
	Alarm:=I140_LK_TST_2_WARNGI704_4 , 
	Endofcycle:=I140_LK_TST_2_END_CYCI704_5,
	StartRSTDly:= , 
	StartOP=>O140_LK_TST2_STRT_Q701_2 , 
	ResetOP=>O140_LK_TST2_RST_Q701_1 ,  
	Receive_String := Ateq_Comm_Prog.sReceived_Data_All[2] ,
	result_Ateq=> OP140_ATEQ2_Result,
	Prg_num=> OP140_ATEQ2_Prgrm_Num,	
    status=> OP140_ATEQ2_Status,	
	Error1=> , 
	Error2=> , 
	Error3=> , 
	ProgSel1=>O140_LK_TST2_SEL1_Q701_3 , 
	ProgSel2=>O140_LK_TST2_SEL2_Q701_4 , 
	ProgSel3=> O140_LK_TST2_SEL3_Q701_5, 
	ProgSel4=> O140_LK_TST2_SEL4_Q701_6, 
	ProgSel5=>O140_LK_TST2_SEL5_Q701_7 , 
	ProgSel6=> O140_LK_TST2_SEL6_Q702_0, 
	ProgSel7=>O140_LK_TST2_SEL7_Q702_1 , 
	ProgSel8=>,
	Result_Completed:=OP140_ATEQ2_ResultCompleted ,
    ResultOK:=OP140_ATEQ2_ResultOK , 
	ResultNOK:= OP140_ATEQ2_ResultNOK );
//ATEQ 3

OP140_ATEQ3_FB(
	AutoSelected:=OP140_AutoSelected , 
	ManualSelected:=OP140_ManualSelected  , 
	Manual_Start:= OP140_ATEQ3_Manual_Start , 
	Auto_Start:= OP140_ATEQ3_Auto_Start , 
	Erroractive:=OP140_ErrorActive , 
	Start:= , 
	Reset:=OP140_ATEQ_Reset  , 
	Manual_Prog_No:=  OP140_ATEQ3_Manual_Prog_No , 
	Auto_Prog_No:=OP140_ATEQ3_Auto_Prog_No_out , 
	Testpass:= I140_LK_TST_3_PASI706_1, 
	Testfail:=I140_LK_TST_3_FLI706_2 , 
	Reffail:=I140_LK_TST_3_REF_PRT_FLI706_3 , 
	Alarm:=I140_LK_TST_3_WARNGI706_4 ,
	Endofcycle:=I140_LK_TST_3_END_CYCI706_5, 
	StartRSTDly:= , 
	StartOP=>O140_LK_TST3_STRT_Q702_3 , 
	ResetOP=>O140_LK_TST3_RST_Q702_2 , 
	
	Receive_String := Ateq_Comm_Prog.sReceived_Data_All[3] ,
	result_Ateq=> OP140_ATEQ3_Result,
	Prg_num=> OP140_ATEQ3_Prgrm_Num,	
    status=> OP140_ATEQ3_Status,	
	Error1=> , 
	Error2=> , 
	Error3=> , 
	ProgSel1=>O140_LK_TST3_SEL1_Q702_4 , 
	ProgSel2=>O140_LK_TST3_SEL2_Q702_5 , 
	ProgSel3=> O140_LK_TST3_SEL3_Q702_6, 
	ProgSel4=> O140_LK_TST3_SEL4_Q702_7, 
	ProgSel5=>O140_LK_TST3_SEL5_Q703_0 , 
	ProgSel6=> O140_LK_TST3_SEL6_Q703_1, 
	ProgSel7=>O140_LK_TST3_SEL7_Q703_2 , 
	ProgSel8=>,
	Result_Completed:=OP140_ATEQ3_ResultCompleted ,
    ResultOK:=OP140_ATEQ3_ResultOK , 
	ResultNOK:= OP140_ATEQ3_ResultNOK );


	//ATEQ 4
	
OP140_ATEQ4_FB(
	AutoSelected:=OP140_AutoSelected , 
	ManualSelected:=OP140_ManualSelected , 
	Manual_Start:= OP140_ATEQ1_Manual_Start , 
	Auto_Start:= OP140_ATEQ4_Auto_Start, 
	Erroractive:=OP140_ErrorActive , 
	Start:= , 
	Reset:=OP140_ATEQ_Reset  , 
	Manual_Prog_No:=  OP140_ATEQ4_Manual_Prog_No , 
	Auto_Prog_No:= OP140_ATEQ4_Auto_Prog_No_out, 
	Testpass:= I140_LK_TST_4_PASI707_1, 
	Testfail:=I140_LK_TST_4_FLI707_2 , 
	Reffail:=I140_LK_TST_4_REF_PRT_FLI707_3 , 
	Alarm:=I140_LK_TST_4_WARNGI707_4 , 
	Endofcycle:=I140_LK_TST_4_END_CYCI707_5,
	StartRSTDly:= , 
	StartOP=>O140_LK_TST4_STRT_Q703_4 , 
	ResetOP=>O140_LK_TST4_RST_Q703_3 , 
	Receive_String := Ateq_Comm_Prog.sReceived_Data_All[4] ,
	result_Ateq=>OP140_ATEQ4_Result,
	Prg_num=> OP140_ATEQ4_Prgrm_Num,	
    status=> OP140_ATEQ4_Status,	
	Error1=> , 
	Error2=> , 
	Error3=> , 
	ProgSel1=>O140_LK_TST4_SEL1_Q703_5 , 
	ProgSel2=>O140_LK_TST4_SEL2_Q703_6 , 
	ProgSel3=> O140_LK_TST4_SEL3_Q703_7, 
	ProgSel4=> O140_LK_TST4_SEL4_Q704_0, 
	ProgSel5=>O140_LK_TST4_SEL5_Q704_1 , 
	ProgSel6=> O140_LK_TST4_SEL6_Q704_2, 
	ProgSel7=>O140_LK_TST4_SEL7_Q704_3 , 
	ProgSel8=>,
	Result_Completed:=OP140_ATEQ4_ResultCompleted,
    ResultOK:=OP140_ATEQ4_ResultOK , 
	ResultNOK:= OP140_ATEQ4_ResultNOK );
	
	
	//ATEQ 5
	
OP140_ATEQ5_FB(
	AutoSelected:=OP140_AutoSelected , 
	ManualSelected:=OP140_ManualSelected  , 
	Manual_Start:= OP140_ATEQ1_Manual_Start , 
	Auto_Start:=OP140_ATEQ5_Auto_Start , 
	Erroractive:=OP140_ErrorActive , 
	Start:= , 
	Reset:=OP140_ATEQ_Reset  , 
	Manual_Prog_No:=  OP140_ATEQ5_Manual_Prog_No , 
	Auto_Prog_No:=OP140_ATEQ5_Auto_Prog_No_out , 
	Testpass:= I140_LK_TST_5_PASI709_3, 
	Testfail:=I140_LK_TST_5_FLI709_4 , 
	Reffail:=I140_LK_TST_5_REF_PRT_FLI709_5 , 
	Alarm:=I140_LK_TST_5_WARNGI709_6 ,
	Endofcycle:=I140_LK_TST_5_END_CYCI709_7,
	StartRSTDly:= , 
	StartOP=>O140_LK_TST5_STRT_Q704_5 , 
	ResetOP=>O140_LK_TST5_RST_Q704_4 ,  
	Receive_String := Ateq_Comm_Prog.sReceived_Data_All[5] ,
	result_Ateq=>OP140_ATEQ5_Result,
	Prg_num=>  OP140_ATEQ5_Prgrm_Num,	
    status=>  OP140_ATEQ5_Status,	
	Error1=> , 
	Error2=> , 
	Error3=> , 
	ProgSel1=> O140_LK_TST5_SEL1_Q704_6 , 
	ProgSel2=> O140_LK_TST5_SEL2_Q704_7 , 
	ProgSel3=> O140_LK_TST5_SEL3_Q705_0, 
	ProgSel4=> O140_LK_TST5_SEL4_Q705_1, 
	ProgSel5=> O140_LK_TST5_SEL5_Q705_2 , 
	ProgSel6=> O140_LK_TST5_SEL6_Q705_3, 
	ProgSel7=> O140_LK_TST5_SEL7_Q705_4 , 
	ProgSel8=> ,
	Result_Completed:=OP140_ATEQ5_ResultCompleted,
    ResultOK:=OP140_ATEQ5_ResultOK , 
	ResultNOK:= OP140_ATEQ5_ResultNOK );

	//ATEQ 6
	
OP140_ATEQ6_FB(
	AutoSelected:=OP140_AutoSelected , 
	ManualSelected:=OP140_ManualSelected  , 
	Manual_Start:= OP140_ATEQ1_Manual_Start , 
	Auto_Start:=OP140_ATEQ6_Auto_Start , 
	Erroractive:=OP140_ErrorActive , 
	Start:= , 
	Reset:=OP140_ATEQ_Reset  , 
	Manual_Prog_No:=  OP140_ATEQ6_Manual_Prog_No , 
	Auto_Prog_No:=OP140_ATEQ6_Auto_Prog_No_out , 
	Testpass:= I140_LK_TST_6_PASI710_1, 
	Testfail:=I140_LK_TST_6_FLI710_2 , 
	Reffail:=I140_LK_TST_6_REF_PRT_FLI710_3 , 
	Alarm:=I140_LK_TST_6_WARNGI710_4 ,
	Endofcycle:=I140_LK_TST_6_END_CYCI710_5, 
	StartRSTDly:= , 
	StartOP=>O140_LK_TST6_STRT_Q705_6 , 
	ResetOP=>O140_LK_TST6_RST_Q705_5 , 
	Receive_String := Ateq_Comm_Prog.sReceived_Data_All[6] ,
	result_Ateq=>OP140_ATEQ6_Result,
	Prg_num=>  OP140_ATEQ6_Prgrm_Num,	
    status=>   OP140_ATEQ6_Status,	
	Error1=> , 
	Error2=> , 
	Error3=> , 
	ProgSel1=> O140_LK_TST6_SEL1_Q705_7 , 
	ProgSel2=> O140_LK_TST6_SEL2_Q706_0 , 
	ProgSel3=> O140_LK_TST6_SEL3_Q706_1, 
	ProgSel4=> O140_LK_TST6_SEL4_Q706_2, 
	ProgSel5=> O140_LK_TST6_SEL5_Q706_3 , 
	ProgSel6=> O140_LK_TST6_SEL6_Q706_4, 
	ProgSel7=> O140_LK_TST6_SEL7_Q706_5 , 
	ProgSel8=>,
	Result_Completed:= OP140_ATEQ6_ResultCompleted,
    ResultOK:=OP140_ATEQ6_ResultOK , 
	ResultNOK:= OP140_ATEQ6_ResultNOK                                               );

END_PROGRAM

// ---- FB/FB/FB/ATEQ_LEAK.TcPOU
FUNCTION_BLOCK ATEQ_LEAK
VAR_INPUT
	AutoSelected: BOOL;
	ManualSelected:BOOL;
	Manual_Start:BOOL;
	Auto_Start:BOOL;
	Erroractive:BOOL;
	Start:BOOL;
	Reset:BOOL;
	Manual_Prog_No:INT;
	Auto_Prog_No:INT;
	Testpass :BOOL;
	Testfail:BOOL;
	Reffail:BOOL;
    Alarm:BOOL;
	Endofcycle:BOOL;
	StartRSTDly:TIME;
	Receive_String : STRING(255);
END_VAR
VAR_OUTPUT
	StartOP:BOOL;
	ResetOP:BOOL;
	
	Error1:BOOL;
	Error2:BOOL;
	Error3:BOOL;
	ProgSel1:BOOL;
	ProgSel2:BOOL;
	ProgSel3:BOOL;
	ProgSel4:BOOL;
	ProgSel5:BOOL;
	ProgSel6:BOOL;
	ProgSel7:BOOL;
	ProgSel8:BOOL;
	result_Ateq,Prg_num,status: STRING(255);		
END_VAR
VAR
Tempend:BOOL;	
TempStart:BOOL;
	ATEQRunning:BOOL;
	ATEQRun: R_TRIG;
	StartResetDly: TON;
	PassTrig: R_TRIG;
	failTrig: R_TRIG;
	Prog_NO:INT;
	Temp_Prog_NO:INT;
	comp:INT;	
	ResetDly: TON;
	EndofcycleTRIG: R_TRIG;
END_VAR

VAR_IN_OUT
	Result_Completed:BOOL;
	ResultOK        :BOOL;
	ResultNOK       :BOOL;
END_VAR

IF (AutoSelected AND Auto_Start)OR (ManualSelected AND Manual_Start) AND NOT Erroractive AND NOT ATEQRunning AND NOT TempStart AND NOT Result_Completed THEN
	ATEQRunning:=TRUE;
	ELSE
		ATEQRunning:=FALSE;
	END_IF
	ATEQRun(CLK:=ATEQRunning , Q=> );
	IF ATEQRun.q AND (Testpass OR Testfail OR Reffail OR Alarm) THEN
		ResetOP:=TRUE;
		Tempend:=FALSE;
	END_IF
	IF ATEQRunning AND (NOT (Testpass OR Testfail OR Reffail OR Alarm) OR ResetDly.Q) THEN
		ResetOP:=FALSE;
	END_IF
	IF ATEQRunning AND NOT ResetOP THEN
		StartOP:=TRUE;
		TempStart:=TRUE;
		ATEQRunning:=FALSE;
			
	END_IF
	
	//IF StartResetDly.Q  THEN
		
	//END_IF
	ResetDly(IN:=ResetOP , PT:=T#500MS , Q=> , ET=> );
	

	PassTrig(CLK:=Testpass , Q=> );
	failTrig(CLK:=Testfail OR  Alarm OR Reffail  , Q=> );
IF EndofcycleTRIG.q THEN 
	Tempend:=TRUE;
END_IF
	IF ( Tempend AND  Testpass ) THEN
		StartOP:=FALSE;	
		ResultOK:=TRUE;
		ResultNOK:=FALSE;
		TempStart:=FALSE;
		Result_Completed:=TRUE;
		Tempend:=FALSE;
		END_IF
IF (Tempend AND (Testfail OR  Reffail OR Alarm)) THEN
	    StartOP:=FALSE;
		ResultNOK:=TRUE;
		ResultOK:=FALSE;
		TempStart:=FALSE;
		Result_Completed:=TRUE;
		Tempend:=FALSE;
		
	END_IF
	
	
	StartResetDly(IN:=StartOP , PT:=T#500MS , Q=> , ET=> );
	
IF (Reset =TRUE)THEN
	ResetOP:=TRUE;
	StartOP:=FALSE;
	TempStart:=FALSE;
	ResultOK:=FALSE;
	ResultNOK:=FALSE;
	ELSE
		ResetOP:=FALSE;
	END_IF
IF ( ManualSelected)THEN
	Temp_Prog_NO:=Manual_Prog_No;

ELSIF(AutoSelected) THEN
	Temp_Prog_NO:=Auto_Prog_No;
	
END_IF
Prog_NO:=Temp_Prog_NO-1;
ProgSel1:=Prog_NO.0;
ProgSel2:=Prog_NO.1;
ProgSel3:=Prog_NO.2;
ProgSel4:=Prog_NO.3;
ProgSel5:=Prog_NO.4;
ProgSel6:=Prog_NO.5;
ProgSel7:=Prog_NO.6;
ProgSel8:=Prog_NO.7;

comp:=FIND(STR1:=Receive_String, STR2:='$R');	
result_Ateq:=MID(STR:=Receive_String, LEN:=(comp-11), POS:=11 );
status:=MID(STR:=Receive_String , LEN:=2, POS:=7 );	
Prg_num:=MID(STR:=Receive_String, LEN:=2, POS:=2 );
EndofcycleTRIG(CLK:=Endofcycle , Q=> );

END_FUNCTION_BLOCK

// ---- POUs/Programs/OP160/OP160_Main.TcPOU
PROGRAM OP160_Main
VAR
	OP160_ModeSelection_FB: Mode_Selection_Block1;
END_VAR

OP160_Error();
OP160_Manual();
OP160_QCPlace_AutoSequence();
OP160_AutoSequence();
OP160_Initialization_Seq();




//ModeSection 

IF (OP160_HMI_AutoMode AND NOT OP160_HMI_ManualMOde AND NOT OP160_HMI_StepMode) THEN
	OP160_Modeselection_FB.ModeWord:=1;
	ELSIF (NOT OP160_HMI_AutoMode AND OP160_HMI_ManualMOde AND NOT OP160_HMI_StepMode) THEN
		OP160_Modeselection_FB.ModeWord:=2;
	ELSIF  (NOT OP160_HMI_AutoMode AND NOT OP160_HMI_ManualMOde AND  OP160_HMI_StepMode) THEN
		OP160_Modeselection_FB.ModeWord:=3;
    ELSE   
		OP160_Modeselection_FB.ModeWord:=0;
END_IF
	






OP160_Modeselection_FB(
	ModeWord:= , 
	HomeConditionOK:=OP160_HomeCondition_OK , 
	OperationEnable:=OperationEnable , 
	StartPB:= , 
	SafetyAndNOError:=OperationEnable , 
	ModeAck:=TRUE , 
	HomingINProgress:= , 
	TempHomeOK:=OP160_Temp_Home_OK , 
	ResetPB:= , 
	AutoSelected=>OP160_AutoSelected , 
	ManualSelected=>OP160_ManualSelected , 
	StepSelected=>OP160_StepSelected , 
	ModeSelAck_Indication=> , 
	StatusDisplay=> , 
	AutoRunning:=OP160_AutoRunning , 
	StepRunning:=OP160_StepRunning , 
	StartEnable:=OP160_StartEnable , 
	MachineStop:=OP160_Machine_Stop );
	
	IF (OP160_AutoSelected OR  OP160_StepSelected ) THEN
		OP160_GVL.OP160_Auto:=TRUE;
		//O160_ROB_MAN_AUTO_MODE_Q709_4:=TRUE;
		OP160_SI_Dry_Run:=TRUE;
		OP160_Robo_Out6002:=1;
		
		ELSE
			OP160_GVL.OP160_Auto:=FALSE;
			//O160_ROB_MAN_AUTO_MODE_Q709_4:=FALSE;
			OP160_Robo_Out6002:=0;
		END_IF
IF OP160_Auto AND NOT OP160_ManualSelected AND NOT OP160_HomeRunning THEN
	OP160_Robo_Out6001:=1;
END_IF
IF OP160_EO_RO_ATC_Open THEN
	O160_TOOL_CHO_UNLOCK_Q1351_0:=TRUE;
	ELSE
		O160_TOOL_CHO_UNLOCK_Q1351_0:=FALSE;
	END_IF
IF OP160_EO_RO_ATC_Close THEN
	O160_TOOL_CHO_LOCK_Q1351_1:=TRUE;
	ELSE
		O160_TOOL_CHO_LOCK_Q1351_1:=FALSE;
	END_IF

END_PROGRAM

// ---- POUs/Programs/OP160/OP160_Error.TcPOU
PROGRAM OP160_Error
VAR
	Step_No: INT;
	AutoStepErr_1: TON;
	OP160_StepErr1: TON;
	OP160_StepErr2: TON;
	bdone: BOOL;
	i: INT;
	j: INT;
END_VAR

IF NOT bdone THEN
	bdone:=TRUE;
FOR i:=1500 TO 1600 BY 1 DO 
	
IF berror[i] THEN
	OP160_ErrorActive:=TRUE;
END_IF
END_FOR
bdone:=FALSE;
END_IF

IF OP130_HMI_Reset OR Servo_Reset THEN
	FOR j:=1500 TO 1600 BY 1 DO 
		
	
	berror[j]:=FALSE;
	OP160_ErrorActive:=FALSE;
	
	END_FOR
	temp:=false;
END_IF

END_PROGRAM

// ---- POUs/Programs/OP160/OP160_Manual.TcPOU
PROGRAM OP160_Manual
VAR
	
	Op160_Robot: FB_Robot;
	OP160_Robo_Automanual_out: BOOL;
	CR160_MoverREM_CylStatus: INT;
	CR160_HMI_Gripper_Cyl_1_Home_PB: BOOL;
	CR160_HMI_Gripper_Cyl_1_Work_PB: BOOL;
	CR160_HMI_Gripper_Cyl_2_Home_PB :BOOL;
	CR160_HMI_Gripper_Cyl_2_Work_PB :BOOL;
	O160_LH_GRPR_OPN_Q1260_5: BOOL;
	O160_LH_GRPR_CLSE_Q1260_4: BOOL;
	OP160_Gripper_Cyl_Status: INT;
	temp5: BOOL;
	temp6: BOOL;
	OP160_GRP_TMR: TON;
	
END_VAR

VAR PERSISTENT
	OP160_GRP_DLY				: TIME;
END_VAR

//Bottom Cylinder 1
CR160_MoverREM_CylStatus:=0;
// Safe Home
IF (TRUE) THEN 
	CR160_MoverREM_Cyl.SafeHome:= TRUE;
	ELSE
		CR160_MoverREM_Cyl.SafeHome:= FALSE;
	END_IF
	//Safe Work
IF(TRUE) THEN 
CR160_MoverREM_Cyl.SafeWork:=TRUE;
ELSE
	CR160_MoverREM_Cyl.SafeWork:=FALSE;
	END_IF
//Manual PB 1
IF(OP160_HMI_MOVREM_Home_PB) THEN
	CR160_MoverREM_Cyl.ManualPB1:=TRUE;
	ELSE
		CR160_MoverREM_Cyl.ManualPB1:=FALSE;
	END_IF
//Manual PB2 
IF(OP160_HMI_MOVREM_Work_PB) THEN
	CR160_MoverREM_Cyl.ManualPB2:=TRUE;
	ELSE
		CR160_MoverREM_Cyl.ManualPB2:=FALSE;
	END_IF	

	

CR160_MoverREM_Cyl(
	Auto:=OP120_AutoSelected , 
	Manual:=OP120_ManualSelected , 
	ErrorActive:=OP160_ErrorActive , 
	ResetPB:=OP160_HMI_Reset , 
	Sensor1:=I160_MOVR_REM_CYL_REVI1311_6 , 
	Sensor2:=I160_MOVR_REM_CYL_FWDI1311_7 , 
	ManualPB1:= , 
	ManualPB2:= , 
	AutoCmd1:= , 
	AutoCmd2:= , 
	OperationEnable:=OperationEnable , 
	SafeHome:= , 
	SafeWork:= , 
	HomingCmd1:= , 
	Pulse_1Sec:=Pulse_Block.Q1Hz , 
	BlinkingBit:= , 
	TimeOut1:=5 , 
	TimeOut2:=5 , 
	TimeOut3:=5 , 
	Solenoid1=> , 
	Solenoid2=>, 
	AlarmSensor1=> , 
	AlarmSensor2=> , 
	AlarmSolenoid1=> , 
	AlarmSolenoid2=> , 
	AllSignal=> , 
	AlarmPresent=> , 
	Position1=> , 
	Position2=> , 
	HomeSensorBlink=> , 
	WorkSensorBlink=> , 
	Status:=CR160_MoverREM_CylStatus );
	
//move ZERO to STATUS
OP120_Gripper_Cyl_Status:=0;



//Reset Auto Cmd IN Manual Mode & Homing
IF (OP160_Auto OR OP160_HomeRunning) THEN
	CR160_Gripper_Cyl_1.AutoCmd1:=FALSE;
	CR160_Gripper_Cyl_1.AutoCmd2:=FALSE;
	CR160_Gripper_Cyl_2.AutoCmd1:=FALSE;
	CR160_Gripper_Cyl_2.AutoCmd2:=FALSE;			
END_IF

// Safe Home
IF (TRUE) AND  (TRUE) THEN 
	CR160_Gripper_Cyl_1.SafeHome:= TRUE ;
	CR160_Gripper_Cyl_2.SafeHome:= TRUE ;
	ELSE 
		CR160_Gripper_Cyl_1.SafeHome:= FALSE ;
		CR160_Gripper_Cyl_2.SafeHome:= FALSE ;
	END_IF
// Safe Work
IF (TRUE) OR (TRUE) THEN 
	CR160_Gripper_Cyl_1.Safework:= TRUE ;
	CR160_Gripper_Cyl_2.Safework:= TRUE ;
	ELSE 
		CR160_Gripper_Cyl_1.Safework:= FALSE ;
		CR160_Gripper_Cyl_2.Safework:= FALSE ;
	END_IF
	
// grippeer 1 Manual PB  Cyl Mapping

IF (CR160_HMI_Gripper_Cyl_1_Home_PB=TRUE OR (OP160_EO_RO_Gripper1_Open AND OP160_ManualSelected)) THEN
	CR160_Gripper_Cyl_1.ManualPB1:=TRUE;
	
		CR160_Gripper_Cyl_1.ManualPB1:=FALSE;
		
	END_IF
	
IF (CR160_HMI_Gripper_Cyl_1_Work_PB=TRUE OR (OP160_EO_RO_Gripper1_Close AND OP160_ManualSelected)) THEN
	
   CR160_Gripper_Cyl_1.ManualPB2:=TRUE;
 
	ELSE 
		
	CR160_Gripper_Cyl_1.ManualPB2:=FALSE;
		
	END_IF

 ////  gripper 2 manual pb cyl mapping 
	
IF (CR160_HMI_Gripper_Cyl_2_Home_PB=TRUE OR (OP160_EO_RO_Gripper2_Open AND OP160_ManualSelected)) THEN
	
	CR160_Gripper_Cyl_2.ManualPB1:=TRUE;
	
	ELSE 
		
		CR160_Gripper_Cyl_2.ManualPB1:=FALSE;
		
	END_IF
	
IF (CR160_HMI_Gripper_Cyl_2_Work_PB=TRUE OR (OP160_EO_RO_Gripper2_Close AND OP160_ManualSelected)) THEN
	
	CR160_Gripper_Cyl_2.ManualPB2:=TRUE;
	
	ELSE 
		
		CR160_Gripper_Cyl_2.ManualPB2:=FALSE;
		
	END_IF	
	
	
	
///////// gripper 1 ////////
	
CR160_Gripper_Cyl_1(
	Auto:=OP160_AutoSelected , 
	Manual:= OP160_ManualSelected, 
	ErrorActive:= OP160_ErrorActive, 
	ResetPB:=OP160_HMI_Reset , 
	Sensor1:=  I160_RH_COMP_PP_GRPR_OPNI712_1  , 
	Sensor2:= NOT I160_RH_COMP_PP_GRPR_OPNI712_1 , 
	ManualPB1:= , 
	ManualPB2:= , 
	AutoCmd1:=OP160_EO_RO_Gripper1_Open AND OP160_AutoSelected , 
	AutoCmd2:=OP160_EO_RO_Gripper1_Close AND OP160_AutoSelected , 
	OperationEnable:=OperationEnable , 
	SafeHome:= , 
	SafeWork:= , 
	HomingCmd1:= , 
	Pulse_1Sec:=Pulse_Block.Q1Hz , 
	BlinkingBit:= , 
	TimeOut1:=5 , 
	TimeOut2:=5 , 
	TimeOut3:=5 , 
	Solenoid1=> , 
	Solenoid2=> , 
	AlarmSensor1=> berror[1506], 
	AlarmSensor2=> berror[1507], 
	AlarmSolenoid1=>berror[1508] , 
	AlarmSolenoid2=>berror[1509] , 
	AllSignal=>berror[1510] , 
	AlarmPresent=> , 
	Position1=> , 
	Position2=> , 
	HomeSensorBlink=> , 
	WorkSensorBlink=> , 
	Status:=OP160_Gripper_Cyl_Status );
	
///// gripper 2///////	

CR160_Gripper_Cyl_2(
	Auto:=OP160_AutoSelected , 
	Manual:= OP160_ManualSelected, 
	ErrorActive:= OP160_ErrorActive, 
	ResetPB:=OP160_HMI_Reset , 
	Sensor1:=  I160_FIXT_LH_COMP_PP_GRPR_OPNI711_7   , 
	Sensor2:= NOT I160_FIXT_LH_COMP_PP_GRPR_OPNI711_7  , 
	ManualPB1:= , 
	ManualPB2:= , 
	AutoCmd1:=OP160_EO_RO_Gripper2_Open AND OP160_AutoSelected , 
	AutoCmd2:=OP160_EO_RO_Gripper2_Close AND OP160_AutoSelected , 
	OperationEnable:=OperationEnable , 
	SafeHome:= , 
	SafeWork:= , 
	HomingCmd1:= , 
	Pulse_1Sec:=Pulse_Block.Q1Hz , 
	BlinkingBit:= , 
	TimeOut1:=5 , 
	TimeOut2:=5 , 
	TimeOut3:=5 , 
	Solenoid1=> , 
	Solenoid2=> , 
	AlarmSensor1=> berror[1511], 
	AlarmSensor2=> berror[1512], 
	AlarmSolenoid1=>berror[1513] , 
	AlarmSolenoid2=>berror[1514] , 
	AllSignal=>berror[1515] , 
	AlarmPresent=> , 
	Position1=> , 
	Position2=> , 
	HomeSensorBlink=> , 
	WorkSensorBlink=> , 
	Status:=OP160_Gripper_Cyl_Status );	
	
	
	IF CR160_Gripper_Cyl_1.Solenoid1 THEN
		O160_LH_COMP_PP_GRPR_CLSE_OPN_Q1350_2:=TRUE;
		//O160_RH_COMP_PP_GRPR_CLSE_OPN_Q1350_3:=TRUE;
	END_IF
	IF CR160_Gripper_Cyl_1.Solenoid2 THEN
		O160_LH_COMP_PP_GRPR_CLSE_OPN_Q1350_2:=FALSE;
		//O160_RH_COMP_PP_GRPR_CLSE_OPN_Q1350_3:=FALSE;
	END_IF	

	IF CR160_Gripper_Cyl_2.Solenoid1 THEN
		//O160_LH_COMP_PP_GRPR_CLSE_OPN_Q1350_2:=TRUE;
		O160_RH_COMP_PP_GRPR_CLSE_OPN_Q1350_3:=TRUE;
	END_IF
	
	IF CR160_Gripper_Cyl_2.Solenoid2 THEN
		//O160_LH_COMP_PP_GRPR_CLSE_OPN_Q1350_2:=FALSE;
		O160_RH_COMP_PP_GRPR_CLSE_OPN_Q1350_3:=FALSE;
	END_IF	
		
///// gripper 1 close fb to robot	
	
IF CR160_Gripper_Cyl_1.Position2 THEN
	OP160_EI_Gripper1_Close:=TRUE;
ELSE
	OP160_EI_Gripper1_Close:=FALSE;
END_IF

///// gripper 1 open fb to robot

IF CR160_Gripper_Cyl_1.Position1 THEN
	OP160_EI_Gripper1_Open:=TRUE;
ELSE
	OP160_EI_Gripper1_Open:=FALSE;
END_IF

///// gripper 2 close fb to robot	
	
IF CR160_Gripper_Cyl_2.Position2 THEN
	OP160_EI_Gripper2_Close:=TRUE;
ELSE
	OP160_EI_Gripper2_Close:=FALSE;
END_IF

///// gripper 2 open fb to robot

IF CR160_Gripper_Cyl_2.Position1 THEN
	OP160_EI_Gripper2_Open:=TRUE;
ELSE
	OP160_EI_Gripper2_Open:=FALSE;
END_IF

OP160_GRP_TMR(IN:=OP160_EO_RO_Gripper1_Close , PT:=OP160_GRP_DLY , Q=> , ET=> );
                	
//RoboFB
				
	Op160_Robot(
	i_b_Operation_Enable_Feedback:= OP160_SO_Auto_Operation_Enable, 
	i_b_Auto_Enable_Feedback:=OP160_SO_Mirror_Auto_enable , 
	i_b_Servo_On_Feedback:= OP160_SO_Servo_ON_OFF_Status, 
	i_b_Servo_Off_Feedback:= OP160_SO_Mirror_SRVO_Off, 
	i_b_Error_Feedback:=OP160_SO_During_error , 
	i_b_Program_Start_Enable_Feedback:=OP160_SO_Program_Execute , 
	i_b_Robo_Stopping_Feedback:=OP160_SO_During_Cycle_Stop , 
	i_b_Emergency_Pressed_Feedback:=OP160_SO_During_EMG_Stop , 
	i_b_Auto_Mode_Feedback:=OP160_SO_Auto_Ext_Mode , 
	i_b_Reset:=OP160_HMI_Reset OR HMI_Reset OR Servo_Reset, 
	i_b_RobotAutoManual:=OP160_Auto , 
	i_b_ProgramReset:=OP160_Robo_ProgramReset , 
	o_b_Operation_Enable_Cmd=>OP160_SI_Operation_Enable , 
	o_b_Auto_Enable_Cmd=>OP160_SI_Auto_Enable , 
	o_b_Servo_On_Cmd=>OP160_SI_Servo_ON , 
	o_b_Servo_Off_Cmd=>OP160_SI_Servo_OFF , 
	o_b_Error_Reset_Cmd=>OP160_SI_Error_Reset , 
	o_b_Program_Reset_Cmd=>OP160_SI_Program_Reset , 
	o_b_Program_Start_Cmd=>OP160_SI_Start , 
	o_b_Program_Stop_Cmd=>OP160_SI_Stop2 , 
	o_b_RobotAutoManual=>OP160_Robo_Automanual_out , 
	o_b_Error=>berror[1550] );

END_PROGRAM

// ---- POUs/Programs/OP160/OP160_QCPlace_AutoSequence.TcPOU
PROGRAM OP160_QCPlace_AutoSequence
VAR
END_VAR



(*
 CASE OP160_AutoPlaceSeq OF
	 10: IF OP160_StartEnable THEN
		 OP160_AutoPlaceSeq:=20;
	 END_IF
	 20:IF OP160_PartPicked AND OP160_StartEnable THEN
		 OP160_AutoPlaceSeq:=30;
	 END_IF
	 30:IF OP160_StartEnable AND OP160_EO_QC_Place_Completed   THEN
		 OP160_Part_Placed:=TRUE;
		 
		  OP160_AutoPlaceSeq:=40;
	 END_IF
	 
	 40:IF OP160_StartEnable THEN
		  OP160_Part_Placed:=FALSE;
		  OP160_AutoPlaceSeq:=50;
	 END_IF
	 50:IF OP160_StartEnable THEN
		 OP160_OperationCompleted:=TRUE;
				 
		  OP160_AutoPlaceSeq:=60;
	 END_IF
	 60:IF OP160_StartEnable THEN
		 OP160_OperationCompleted:=FALSE;
		 OP160_PartPicked:=FALSE;
		 OP160_AutoPlaceSeq:=10;
	 END_IF
 END_CASE 
*)

END_PROGRAM

// ---- POUs/Programs/OP160/OP160_AutoSequence.TcPOU
PROGRAM OP160_AutoSequence
VAR
	OP160_AutoSeq:INT;
	OP160_MoverinstationTRIG				: R_TRIG;
	dllt: ton;
	COMPLETE_R_TRIG: R_TRIG;
	fix_lh_1: INT;
	fix_rh_1: INT;
	dry_run :bool;
END_VAR

IF (NOT OP160_Auto OR  OP160_ErrorActive OR OP160_HomeRunning OR OP160_Machine_Stop ) THEN
	
	OP160_AutoRunning               := FALSE;
	OP160_ComponentOk               :=FALSE;
	OP160_ComponentNok              :=FALSE;
	OP160_Moverpresent              :=FALSE;
	op160_place_both_component_ok   :=FALSE;
	op160_place_1_ok_1_nok          :=FALSE;
	op160_go_to_place               :=FALSE;
    op160_place_both_component_rej  := FALSE;
	OP160_AutoPlaceSeq              :=0;
	OP160_AutoSeq                   := 10;
	OP160_Prev_LH_COMP_OK           := FALSE;
    OP160_Prev_RH_COMP_OK           := FALSE;
	op160_comp_Lh_ok_to_rbt         := FALSE;
	op160_comp_Lh_nok_to_rbt        := FALSE;
	op160_comp_rh_ok_to_rbt         := FALSE;
	op160_comp_rh_nok_to_rbt        := FALSE;
	OP160_PartPicked                :=FALSE;
END_IF

CASE OP160_AutoSeq OF 
	10:IF (OP160_Auto) THEN		// Check Automode Selected
		OP160_AutoSeq :=20;
	    END_IF
	20:IF ( NOT OP160_ErrorActive) THEN		//Check No error
		OP160_AutoSeq:=30;
	   END_IF
	30:IF (NOT OP160_HomeRunning) THEN		//Check No Homerunning
		OP160_AutoSeq :=40;
		END_IF
    40:IF ( OP160_Temp_Home_OK)THEN	//Check Machine in Home
		OP160_AutoSeq:= 50;
		END_IF
	50:IF ( NOT OP160_OperationCompleted) THEN		// Check Operation Completed Reset
		OP160_AutoSeq:=60;
		END_IF
		
	60:IF (NOT OP160_ComponentOk) THEN		// Check Component Ok Reset
		OP160_AutoSeq:=70;
		END_IF
		
	70:IF (NOT OP160_ComponentNok) THEN 	// Check Component NOk Reset
		OP160_AutoSeq:= 120;
		OP160_AutoPlaceSeq:=10;
		END_IF
		
		
    120:IF  ( OP160_HMI_Cycle_Start ) THEN		//Machine Start in Fully Automatic or Press Cycle Start For Semi Automatic
		    OP160_HomeCondition_OK:=TRUE;
	 			IF( OP160_HomeCondition_OK AND OP160_AutoSelected) THEN
					OP160_AutoRunning:=TRUE;
					OP160_StepRunning:= FALSE;
				
				ELSIF ( OP160_HomeCondition_OK AND OP160_StepSelected) THEN
					OP160_AutoRunning:=FALSE;
					OP160_StepRunning:= TRUE;
				END_IF;
		 END_IF
		 IF ((OP160_AutoRunning OR OP160_StepRunning) AND OP160_StartEnable) THEN
			 		O160_VFD_FWD_Q708_0  :=1;
		            O160_VFD_STOP_Q708_2 :=1;
					OP160_Prev_Comp_Status:=1;
					OP160_AutoSeq:= 140;
		END_IF
		
	140: IF  OP160_StartEnable AND OP160_STN_ENABLE  THEN
                IF fix_lh_1 >0 AND fix_rh_1 >0 THEN
		           OP160_Prev_LH_COMP_OK           := TRUE;
	               OP160_Prev_RH_COMP_OK           := TRUE;
				   
				   op160_comp_Lh_ok_to_rbt         := TRUE;
	               op160_comp_Lh_nok_to_rbt        := FALSE;
	               op160_comp_rh_ok_to_rbt         := TRUE;
	               op160_comp_rh_nok_to_rbt        := FALSE; 
				   
   		           OP160_AutoSeq := 150;
																																																																																				
		        ELSIF fix_lh_1 =158 AND fix_rh_1 =159 THEN
					
		        	  OP160_Prev_LH_COMP_OK           := TRUE;
	                  OP160_Prev_RH_COMP_OK           := FALSE;
					  
					  op160_comp_Lh_ok_to_rbt         := TRUE;
					  op160_comp_Lh_nok_to_rbt        := FALSE;
					  op160_comp_rh_ok_to_rbt         := FALSE;
					  op160_comp_rh_nok_to_rbt        := TRUE;  
			
		        	  OP160_AutoSeq := 150;
					  
		        ELSIF fix_lh_1 =159 AND fix_rh_1 =158 THEN
		        	  OP160_Prev_LH_COMP_OK           := FALSE;
	                  OP160_Prev_RH_COMP_OK           :=TRUE ;
					  
                      op160_comp_Lh_ok_to_rbt         := FALSE;
                      op160_comp_Lh_nok_to_rbt        := TRUE;
                      op160_comp_rh_ok_to_rbt         := TRUE;
                      op160_comp_rh_nok_to_rbt        := FALSE;  
  
	                  OP160_AutoSeq := 150;
					  
	            ELSIF  fix_lh_1 =159 AND fix_rh_1 =159 THEN
	                   OP160_Prev_LH_COMP_OK           := FALSE;
		               OP160_Prev_RH_COMP_OK           :=FALSE ;
					   
					   op160_comp_Lh_ok_to_rbt         := FALSE;
					   op160_comp_Lh_nok_to_rbt        := TRUE;
					   op160_comp_rh_ok_to_rbt         := FALSE;
					   op160_comp_rh_nok_to_rbt        := TRUE; 
					   
                       OP160_AutoSeq := 150;  
		        END_IF
				END_IF
		
	150:       IF OP160_StartEnable  THEN
		          OP160_Moverpresent                   :=TRUE;
		          OP160_AutoSeq                        := 151;
	           END_IF
			   
	151: COMPLETE_R_TRIG(CLK:=OP160_EO_QC_Pick_Completed , Q=> );
         IF COMPLETE_R_TRIG.Q THEN
		    OP160_PartPicked                           :=TRUE;
          END_IF
		  IF OP160_PartPicked THEN
	           IF  OP160_Prev_LH_COMP_OK AND OP160_Prev_RH_COMP_OK THEN
				   op160_place_both_component_ok       := TRUE;
					OP160_AutoSeq                      := 152;
					
			   ELSIF (NOT OP160_Prev_LH_COMP_OK AND  OP160_Prev_RH_COMP_OK) OR ( OP160_Prev_LH_COMP_OK AND NOT OP160_Prev_RH_COMP_OK) THEN
                     // op160_place_1_ok_1_nok           := TRUE;
					  op160_go_to_place                := TRUE;
					  OP160_AutoSeq                    := 153;
					  
			   ELSIF NOT OP160_Prev_LH_COMP_OK AND NOT OP160_Prev_RH_COMP_OK THEN
	                     op160_place_both_component_rej:= TRUE;
						 OP160_AutoSeq:= 154;
			   END_IF
		     END_IF

    152: IF op160_place_both_component_ok AND OP160_EO_QC_Place_Completed THEN
		    op160_place_both_component_ok               := FALSE;
            OP160_AutoSeq                               := 160;
	     END_IF


	153: IF OP160_EO_QC_Place_Completed AND op160_go_to_place THEN
			op160_place_1_ok_1_nok                      := TRUE ; 
			op160_go_to_place                           := FALSE;
			OP160_AutoSeq                               := 155;  
	    END_IF		
			
			
	     
		 
	154: IF op160_place_both_component_rej AND OP160_EO_Rejection_Place_Completed THEN
			op160_place_both_component_rej              :=FALSE;	
			OP160_AutoSeq                               := 160;	
	     END_IF
	
    155: IF  op160_place_1_ok_1_nok AND OP160_EO_Rejection_Place_Completed THEN
			 //  op160_go_to_place                        := FALSE;
			   op160_place_1_ok_1_nok                   := FALSE ;
               OP160_AutoSeq                            := 160; 
		END_IF
	
	160:    OP160_Moverpresent                         :=FALSE;
		    OP160_AutoSeq                              := 170;	   
		       

	170: OP160_AutoSeq                                 := 180;
		       
		
	180:       IF OP160_StartEnable AND NOT OP160_SO_Rbt_In_Pick_Zone AND NOT I160_FIXT_COMP1_PRSNI1320_4 AND NOT I160_FIXT_COMP1_PRSNI1320_4 THEN 
		          STATION_DONE[OP160_STN_MOVER][OP160_XTS_POS_NO]			:= TRUE;
		          MOVER_CMP_STATUS[OP160_STN_MOVER][2]:=0;
		          MOVER_CMP_STATUS[OP160_STN_MOVER][1]:=0;
		          OP160_AutoSeq:= 250;
		       END_IF
		
	
	250:       // Reset All Bits							
               OP160_LH_Comp_OK:=FALSE;
               OP160_LH_Comp_NOK:=FALSE;
               OP160_RH_Comp_OK:=FALSE;
               OP160_RH_Comp_NOK:=FALSE;
			   OP160_Prev_LH_COMP_OK := FALSE;
			   OP160_Prev_RH_COMP_OK := FALSE;
			   OP160_PartPicked      :=FALSE;
			   op160_comp_Lh_ok_to_rbt         := FALSE;
			   op160_comp_Lh_nok_to_rbt        := FALSE;
			   op160_comp_rh_ok_to_rbt         := FALSE;
			   op160_comp_rh_nok_to_rbt        := FALSE;
               OP160_AutoSeq    := 120;
				
		
END_CASE

OP160_EI_Camera_OK :=TRUE;
OP160_MoverinstationTRIG(CLK:=OP160_MoverinStation , Q=> );
dry_run:=All_Station_Dry_Run;
IF Dry_Run THEN
	fix_lh_1:=158;	
    fix_rh_1:=158;
ELSE
	fix_lh_1:=MOVER_CMP_STATUS[OP160_STN_MOVER][1];	
    fix_rh_1:=MOVER_CMP_STATUS[OP160_STN_MOVER][2];	
END_IF

//############################		OP160 STATION ENABLE CONDITION		##########################

	OP160_STN_MOVER					:= MOVER_POSITION[OP160_XTS_POS_NO];
	IF AUTO_WITH_XTS THEN
	IF OP160_STN_MOVER>0 THEN
	IF NOT(END_OF_CYCLE AND MOVER_CMP_STATUS[OP160_STN_MOVER][1]=5 AND MOVER_CMP_STATUS[OP160_STN_MOVER][2]=5)THEN
	OP160_STN_ENABLE					:= MOVER_POS_RECHED[OP160_STN_MOVER] AND ((MOVER_CMP_STATUS[OP160_STN_MOVER][1]>0)OR 
										(MOVER_CMP_STATUS[OP160_STN_MOVER][2]>0)) AND STATION_ENABLE_CONTROL;	
	ELSE
	STATION_DONE[OP160_STN_MOVER][OP160_XTS_POS_NO]			:= TRUE;		
	END_IF
	ELSE
	OP160_STN_ENABLE					:= FALSE;	
	END_IF	
	END_IF

END_PROGRAM

// ---- POUs/Programs/OP160/OP160_Initialization_Seq.TcPOU
PROGRAM OP160_Initialization_Seq
VAR
	op160_master_reset :BOOL;
	op160_robot_homed  :BOOL;
	op160_ROboProgResetDly   :ton;
END_VAR

IF CR160_MoverREM_Cyl.Position1 AND OP160_SO_Rbt_In_Home AND op160_robot_homed THEN
   OP160_Temp_Home_OK:=TRUE;
ELSE
	OP160_Temp_Home_OK:=FALSE;
END_IF

IF OP160_ErrorActive THEN 
	op160_robot_homed    :=FALSE;
END_IF

CASE OP160_Homing_Seq OF
	
	0: IF (OP160_Auto AND NOT OP160_HomeRunning AND  NOT OP160_ErrorActive AND  NOT 
			OP160_AutoRunning AND NOT OP160_StepRunning	 AND NOT OP160_Temp_Home_OK) THEN
		    OP160_HomeRunning:=TRUE;
		    OP160_Homing_Seq:=10;	
	   END_IF
	   
	10:IF (OP160_HomeRunning AND OP160_HMI_Homing)THEN
		OP160_Homing_Seq:=12;		
		END_IF 
        
	
   12:  OP160_Robo_ProgramReset:=TRUE;
   
		IF NOT OP160_SO_Program_Execute	AND op160_ROboProgResetDly.Q THEN
		OP160_Robo_ProgramReset:=FALSE;			
		OP160_Homing_Seq:=14;	
		END_IF
	
		
	
	14: IF OP160_HomeRunning AND NOT op160_master_reset THEN
		   OP160_Robo_Out6001   :=1;
	       OP160_SI_Homing_Start:=TRUE;
	       OP160_Homing_Seq:=15;
	    
		ELSIF  OP160_HomeRunning AND  op160_master_reset THEN
		       OP160_Robo_Out6001   :=3;
	           OP160_SI_Homing_Start:=TRUE;
	           OP160_Homing_Seq     :=15;
		END_IF
		
		
      (*  OP160_Robo_Out6001:=3;
        
		IF OP160_SO_Rbt_In_Home THEN
		OP160_SI_Homing_Start:=FALSE;
		
		OP160_Robo_ProgramReset:=TRUE;	
		END_IF
		IF NOT OP160_SO_Program_Execute	AND OP160_Robo_ProgramReset=TRUE THEN
		OP160_Robo_ProgramReset:=FALSE;
		OP160_Homing_Seq:=20;		
		END_IF *)
			
	15: IF OP160_HomeRunning AND OP160_SO_Rbt_In_Home THEN
		   OP160_SI_Homing_Start:=FALSE;
		   op160_robot_homed    :=TRUE;
		   OP160_Homing_Seq:=20;
	    END_IF
 
	
	20:IF (OP160_HomeRunning AND OP160_HMI_Homing)THEN 
        IF ( CR160_MoverREM_Cyl.Position1 ) THEN
			OP160_Homing_Seq:=30;
		ELSE
			CR160_MoverREM_Cyl.HomingCmd1:= TRUE;
				
		END_IF
		END_IF
	
		
	30:	OP160_Homing_Seq:=0;
		OP160_HomeRunning:=FALSE;
	
END_CASE

IF NOT OP160_HomeRunning THEN
	CR160_MoverREM_Cyl.HomingCmd1:= FALSE;
END_IF

op160_ROboProgResetDly(IN:= OP160_Robo_ProgramReset, PT:= T#200MS, Q=> , ET=> );

END_PROGRAM

// ---- POUs/GENERAL/IO_Diag.TcPOU
PROGRAM IO_Diag
VAR
	Panel_num : INT := 1;
	i : UINT;
	j : UINT;
	Input_Page_num : UINT;
	Output_Page_num : UINT;
	
	IP_Arr_OP10A : ARRAY[0..100] OF UINT := [100,101,102,103];
	OP_Arr_OP10A : ARRAY[0..100] OF UINT := [100,101,102,103];
	IP_Arr_OP10B : ARRAY[0..100] OF UINT := [200,201,202,203];
	OP_Arr_OP10B_JB : ARRAY[0..100] OF UINT := [200,201,202,203];
	IP_Arr_OP10P : ARRAY[0..100] OF UINT := [302,303,304,305,306,307,308,309,310,311,1000,1001,1010,1011,1020,1021,1030,1031,1040,1041,1100,1101,1110,1111]; 
	OP_Arr_OP10P : ARRAY[0..100] OF UINT := [300,301,302,303,304,305,306,307,308,309,1050,1051,1052,1053,1060,1061,1062,1063,1150,1151,1152,1153];
	IP_Arr_OP90P : ARRAY[0..100] OF UINT := [400,401,402,403,404,405,1200,1201,1210,1211,1220,1221];
	OP_Arr_OP90P : ARRAY[0..100] OF UINT := [400,401,402,403,1240,1241,1242,1250,1251,1260,1261,1262];
	IP_Arr_OP160P : ARRAY[0..100] OF UINT := [700,701,702,703,704,705,706,707,708,709,710,711,712,713,714,715,1300,1301,1310,1311,1320,1321,1330,1331];
	OP_Arr_OP160P : ARRAY[0..100] OF UINT := [700,701,702,703,704,705,706,707,708,709,1340,1341,1342,1343,1350,1351,1352,1353];
	IP_Arr_OP90JB : ARRAY[0..100] OF UINT := [500,501,502,503,504,505];
	OP_Arr_OP90 : ARRAY[0..100] OF UINT := [500,501,502,503];	
	IP_Arr_OP120_JB : ARRAY[0..100] OF UINT := [600,601,602,603];
	OP_Arr_OP120 : ARRAY[0..100] OF UINT := [600,601,602,603];
	Safety_IP    : ARRAY[0..100] OF UINT := [400,401,402,700];
	Safety_OP    : ARRAY[0..100] OF UINT := [400,700];
	
    Line1: WSTRING;
	Line2: WSTRING;	
	Line3: WSTRING;
	Line4: WSTRING;
	Line5: WSTRING;
	Line6: WSTRING;
	Line7: WSTRING;
	Line8: WSTRING;
	
	OLine1: WSTRING;
	OLine2: WSTRING;
	OLine3: WSTRING;
	OLine4: WSTRING;
	OLine5: WSTRING;
	OLine6: WSTRING;
	OLine7: WSTRING;
	OLine8: WSTRING;

	Lamp1 : BOOL;
	Lamp2 : BOOL;
	Lamp3 : BOOL;
	Lamp4 : BOOL;
	Lamp5 : BOOL;
	Lamp6 : BOOL;
	Lamp7 : BOOL;
	Lamp8 : BOOL;
	
	Visibility_1 : BOOL;
	Visibility_2 : BOOL;
	Visibility_3 : BOOL;
	Visibility_4 : BOOL;
	Visibility_5 : BOOL;
	Visibility_6 : BOOL;
	Visibility_7 : BOOL;
	Visibility_8 : BOOL;
	
	Out_Lamp1 : BOOL;
	Out_Lamp2 : BOOL;
	Out_Lamp3 : BOOL;
	Out_Lamp4 : BOOL;
	Out_Lamp5 : BOOL;
	Out_Lamp6 : BOOL;
	Out_Lamp7 : BOOL;
	Out_Lamp8 : BOOL;
	
	Out_Visibility_1 : BOOL;
	Out_Visibility_2 : BOOL;
	Out_Visibility_3 : BOOL;
	Out_Visibility_4 : BOOL;
	Out_Visibility_5: BOOL;
	Out_Visibility_6: BOOL;
	Out_Visibility_7 : BOOL;
	Out_Visibility_8 : BOOL;
	
	
	Out_Visibility: BOOL;

END_VAR

CASE panel_num OF 
 1: CASE IP_Arr_OP10P[Input_Page_num] OF
   //300: Line1:= "I10A_SPARE_I300_0(I300.0) "                   ;
   //301: Line1:= "I10A_SPARE_I301_0(I301.0) "                   ;
     302: Line1:= "I10B_DRUM_FEED_ALRM(I302.0)"                  ;
     303: Line1:= "I10B_SPARE_I303_0(I303.0)  "                  ;
     304: Line1:= "I30_DRUM_FEED_ALRM(I304.0) "                  ;
     305: Line1:= "I40_ATC_DECLAMP_FB(I305.0) "                  ;
     306: Line1:= "I50_DRUM_FEED_ALRM(I306.0) "                  ;
     307: Line1:= "I60_ATC_DECLAMP_FB(I307.0) "                  ;
     308: Line1:= "I70_DRUM_FEED_ALRM(I308.0) "                  ;
     309: Line1:= "I80_ATC_DECLAMP_FB(I309.0) "                  ;
     310: Line1:= "I80_SPARE_I310.0(I310.0) "                    ;
     311: Line1:= "I80_SPARE_I311.0(I311.0) "                    ;
     1000: Line1:= "I10A_MAIN_AIR_PRES_FB(I1000.0) "             ;
     1001: Line1:= "I10A_SPARE_I1001_0(I1001.0) "              ;
     1010: Line1:= "I10A_DRUM_LH_CONV_OVR_FLW(I1010.0) "         ;
     1011: Line1:= "I10A_ORING_ROTRY_CYL_O_DEG(I1011.0) "        ;
     1020: Line1:= "I10A_RH_FIRTRE_ORING_REJ_CYL_REV(I1020.0) "  ;
     1021: Line1:= "I10A_BOWL_TRK_INDXR_POS2(I1021.0) "          ;
     1030: Line1:= "I10B_DRUM_LH_CONV_OVR_FLW(I1030.0) "         ;
     1031: Line1:= "I10B_ORING_ROTRY_CYL_O_DEG(I1031.0) "        ;
     1040: Line1:= "I10B_RH_FIRTRE_ORING_REJ_CYL_REV(I1040.0) "  ;
     1041: Line1:= "I10B_BOWL_TRK_INDXR_POS2(I1041.0) "          ;
     1100: Line1:= "I30_DRUM_FEED_CONV1_OVERFL(I1100.0) "        ;
     1101: Line1:= "I50_DRUM_FEED_CONV1_OVERFLW(I1101.0) "       ;
     1110: Line1:= "I50_SPARE_I1110_0(I1110.0) "                 ;
     1111: Line1:= "I50_TOP_REJ_BIN_PRSNCE(I1111.0) "            ;
     
     ELSE
       Line1:= " ";	
     END_CASE
	 Visibility_1:=TRUE;
   
     CASE IP_Arr_OP10P[Input_Page_num] OF
	      //300: Lamp1:=I10A_SPARE_I300_0                    ;
              //301: Lamp1:=I10A_SPARE_I301_0                    ;
		302: Lamp1:=I10B_DRUM_FEED_ALRM_I302_0           ;
		303: Lamp1:=I10B_SPARE_I303_0 			 ;
		304: Lamp1:=I30_DRUM_FEED_ALRM_I304_0  		 ;
		305: Lamp1:=I40_ATC_DECLAMP_FB_I305_0 		 ;
		306: Lamp1:=I50_DRUM_FEED_ALRM_I306_0            ;
		307: Lamp1:=I60_ATC_DECLAMP_FB_I307_0            ;
		308: Lamp1:=I70_DRUM_FEED_ALRM_I308_0            ;
		309: Lamp1:=I80_ATC_DECLAMP_FB_I309_0            ;
		310: Lamp1:=I80_SPARE_I310_0                     ;
		311: Lamp1:=I80_SPARE_I311_0                     ;
		1000: Lamp1:=I10A_MAIN_AIR_PRES_FB_I1000_0       ;
		1001: Lamp1:=I10_LH_LNR_TRCK_FIX_CHO_2_I1001_0 ;
		1010: Lamp1:=I10A_DRUM_LH_CONV_OVR_FLW_I1010_0   ;
		1011: Lamp1:=I10A_ORING_ROTRY_CYL_O_DEG_I1011_0  ;
		1020: Lamp1:=I10A_RH_FIRTRE_ORING_REJ_CYL_REV_I1020_0 ;
		1021: Lamp1:=I10A_BOWL_TRK_INDXR_POS2_I1021_0    ;
		1030: Lamp1:=I10B_DRUM_LH_CONV_OVR_FLW_I1030_0   ;
		1031: Lamp1:=I10B_ORING_ROTRY_CYL_O_DEG_I1031_0  ;
		1040: Lamp1:=I10B_RH_FIRTRE_ORING_REJ_CYL_REV_I1040_0 ;
		1041: Lamp1:=I10B_BOWL_TRK_INDXR_POS2_I1041_0    ;
		1100: Lamp1:=I30_DRUM_FEED_CONV1_OVERFLW_I1100_0 ;
		1101: Lamp1:=I50_DRUM_FEED_CONV1_OVERFLW_I1101_0 ;
		1110: Lamp1:=I50_SPARE_I1110_0;
		1111: Lamp1:=I50_TOP_REJ_BIN_PRSNCE_I1111_0 ;
     ELSE
       Visibility_1:=FALSE;	
     END_CASE
	 
     CASE IP_Arr_OP10P[Input_Page_num] OF
     //300: Line2:=  "I10A_SPARE_I300_1(I300.1)"              ;
     //301: Line2:=  "I10A_SPARE_I301_1(I301.1)"              ;
     302: Line2:=  "I10A_SPARE_I302_1(I302.1)"                ;
     303: Line2:=  "I10B_SPARE_I303_1(I303.1)"                ;
     304: Line2:=  "I30_SPARE_I304_1(I304.1) "                ;
     305: Line2:=  "I40_ATC_CLAMP_FB(I305.1) "                ;
     306: Line2:=  "I50_SPARE_I306_1(I306.1) "                ;
     307: Line2:=  "I60_ATC_CLAMP_FB(I307.1) "                ;
     308: Line2:=  "I70_SPARE_I308_1(I308.1) "                ;
     309: Line2:=  "I80_ATC_CLAMP_FB(I309.1) "                ;
     310: Line2:=  "I80_SPARE_I310_1(I310.1) "                ;
     311: Line2:=  "I80_SPARE_I311_1(I311.1) "                ;
     1000: Line2:= "I10A_SPARE_I1000_1(I1000.1) "             ;
     1001: Line2:= "I10A_SPARE_I1001,1(I1001,1) "           ;
     1010: Line2:= "I10A_DRUM_RH_CONV_OVR_FLW(I1010.1)"       ;
     1011: Line2:= "I10A_ORING_ROTRY_CYL_180_DEG(I1011.1)  "  ;
     1020: Line2:= "I10A_RH_FIRTRE_ORING_REJ_CYL_FWD(I1020.1)";
     1021: Line2:= "I10A_BOWL_TRK_INDXR_POS3(I1021.1) "       ;
     1030: Line2:= "I10B_DRUM_RH_CONV_OVR_FLW(I1030.1)"       ;
     1031: Line2:= "I10B_ORING_ROTRY_CYL_180_DEG(I1031.1)  "  ;
     1040: Line2:= "I10B_RH_FIRTRE_ORING_REJ_CYL_FWD(I1040.1)";
     1041: Line2:= "I10B_BOWL_TRK_INDXR_POS3(I1041.1)  "      ;
     1100: Line2:= "I30_DRUM_FEED_CONV2_OVERFLW(I1100.1) "    ;
     1101: Line2:= "I50_DRUM_FEED_CONV2_OVERFLW(I1101.1) "    ;
     1110: Line2:= "I50_RH_GRIP_CLSE(I1110.1) "               ;
     1111: Line2:= "I50_BOT_REJ_BIN_PRSNCE_I1111_1(I1111.1) " ;
     ELSE
     	Line2 := " ";
     END_CASE
	 
	 Visibility_2:=TRUE;
     CASE IP_Arr_OP10P[Input_Page_num] OF
	//300: Lamp2:=I10A_SPARE_I300_1 ;
	//301: Lamp2:=I10A_SPARE_I301_1 ;
	302: Lamp2:=I10A_SPARE_I302_1 ;
	303: Lamp2:=I10B_SPARE_I303_1 ;
	304: Lamp2:=I30_SPARE_I304_1 ;
	305: Lamp2:=I40_ATC_CLAMP_FB_I305_1 ;
	306: Lamp2:=I50_SPARE_I306_1 ;
	307: Lamp2:=I60_ATC_CLAMP_FB_I307_1 ;
	308: Lamp2:=I70_SPARE_I308_1 ;
	309: Lamp2:=I80_ATC_CLAMP_FB_I309_1 ;
	310: Lamp2:=I80_SPARE_I310_1 ;
	311: Lamp2:=I80_SPARE_I311_1 ;
	1000: Lamp2:=I10A_SPARE_I1000_1 ;
	1001: Lamp2:=I10_RH_LNR_TRCK_FIX_CHO_1_I1001_1 ;
	1010: Lamp2:=I10A_DRUM_RH_CONV_OVR_FLW_I1010_1 ;
	1011: Lamp2:=I10A_ORING_ROTRY_CYL_180_DEG_I1011_1 ;
	1020: Lamp2:=I10A_RH_FIRTRE_ORING_REJ_CYL_FWD_I1020_1 ;
	1021: Lamp2:=I10A_BOWL_TRK_INDXR_POS3_I1021_1;
	1030: Lamp2:=I10B_DRUM_RH_CONV_OVR_FLW_I1030_1  ;
	1031: Lamp2:=I10B_ORING_ROTRY_CYL_180_DEG_I1031_1  ;
	1040: Lamp2:=I10B_RH_FIRTRE_ORING_REJ_CYL_FWD_I1040_1  ;
	1041: Lamp2:=I10B_BOWL_TRK_INDXR_POS3_I1041_1  ;
	1100: Lamp2:=I30_DRUM_FEED_CONV2_OVERFLW_I1100_1  ;
	1101: Lamp2:=I50_DRUM_FEED_CONV2_OVERFLW_I1101_1  ;
	1110: Lamp2:=I50_RH_GRIP_CLSE_I1110_1 ;
	1111: Lamp2:=I50_BOT_REJ_BIN_PRSNCE_I1111_1 ;
   ELSE
       Visibility_2:=FALSE;	
   END_CASE 
   
     CASE IP_Arr_OP10P[Input_Page_num] OF
     //300:  Line3:= "I10A_SPARE_I300_2(I300.2)               "  ;
     //301:  Line3:= "I10A_SPARE_I301_2(I301.2)               "  ;
     302:  Line3:= "I10B_DRUM_OFF_ON(I302.2)                  "  ;
     303:  Line3:= "I10B_SPARE_I303_2(I303.2)                 "  ;
     304:  Line3:= "I30_DRUM_OFF_ON(I304.2)                   "  ;
     305:  Line3:= "I40_ATC_STN_POKE_YOKE_1(I305.2)           "  ;
     306:  Line3:= "I50_DRUM_OFF_ON(I306.2)                   "  ;
     307:  Line3:= "I60_ATC_STN_POKE_YOKE_1(I307.2)           "  ;
     308:  Line3:= "I70_DRUM_OFF_ON(I308.2)                   "  ;
     309:  Line3:= "I80_ATC_STN_POKE_YOKE_1(I309.2)           "  ;
     310:  Line3:= "I80_SPARE_I310_2(I310.2)                  "  ;
     311:  Line3:= "I80_SPARE_I311_2(I311.2)                  "  ;
     1000: Line3:= "I10A_BDY_REJ_BIN_OVERFLW(I1000.2)         "  ;
     1001: Line3:= "I10A_SPARE_I1001,2(I1001,2)             "  ;
     1010: Line3:= "I10A_ORING_LH_GRPR_CLSE(I1010.2)          "  ;
     1011: Line3:= "I10A_ORING_HORZ_CYL_REV(I1011.2)          "  ;
     1020: Line3:= "I10A_BDY_SING_CYL_CLSE(I1020.2)           "  ;
     1021: Line3:= "I10A_SPARE_I1021_2(I1021.2)               "  ;
     1030: Line3:= "I10B_ORING_LH_GRPR_CLSE(I1030.2)          "  ;
     1031: Line3:= "I10B_ORING_HORZ_CYL_REV(I1031.2)          "  ;
     1040: Line3:= "I10B_BDY_SING_CYL_CLSE(I1040.2)           "  ;
     1041: Line3:= "I10B_SPARE_I1041_2(I1041.2)               "  ;
     1100: Line3:= "I30_LH_REJ_CYL_FWD(I1100.2)               "  ;
     1101: Line3:= "I50_LH_REJ_CYL_FWD(I1101.2)               "  ;
     1110: Line3:= "I70_DRUM_FEED_CONV1_OVERFLW(I1110.2)      "  ;
     1111: Line3:= "I70_TOP_REJ_BIN_PRSNCE_I1111_2(I1111.2)   "  ;  
     ELSE
     	Line3 := " ";
     END_CASE
	 
	Visibility_3:=TRUE;
    CASE IP_Arr_OP10P[Input_Page_num] OF
	//300: Lamp3:=I10A_SPARE_I300_2 ;
	//301: Lamp3:=I10A_SPARE_I301_2 ;
	302: Lamp3:=I10B_DRUM_OFF_ON_I302_2 ;
	303: Lamp3:=I10B_SPARE_I303_2 ;
	304: Lamp3:=I30_DRUM_OFF_ON_I304_2 ;
	305: Lamp3:=I40_ATC_STN_POKE_YOKE_1_I305_2 ;
	306: Lamp3:=I50_DRUM_OFF_ON_I306_2 ;
	307: Lamp3:=I60_ATC_STN_POKE_YOKE_1_I307_2 ;
	308: Lamp3:=I70_DRUM_OFF_ON_I308_2;
	309: Lamp3:=I80_ATC_STN_POKE_YOKE_1_I309_2;
	310: Lamp3:=I80_SPARE_I310_2  ;
	311: Lamp3:=I80_SPARE_I311_2  ;
	1000: Lamp3:=I10A_BDY_REJ_BIN_OVERFLW_I1000_2 ;
	1001: Lamp3:=I10_RH_LNR_TRCK_FIX_CHO_2_I1001_2;
	1010: Lamp3:=I10A_ORING_LH_GRPR_CLSE_I1010_2 ;
	1011: Lamp3:=I10A_ORING_HORZ_CYL_REV_I1011_2;
	1020: Lamp3:=I10A_BDY_SING_CYL_CLSE_I1020_2;
	1021: Lamp3:=I10A_SPARE_I1021_2 ;
	1030: Lamp3:=I10B_ORING_LH_GRPR_CLSE_I1030_2  ;
	1031: Lamp3:=I10B_ORING_HORZ_CYL_REV_I1031_2  ;
	1040: Lamp3:=I10B_BDY_SING_CYL_CLSE_I1040_2 ;
	1041: Lamp3:=I10B_SPARE_I1041_2 ;
	1100: Lamp3:=I30_LH_REJ_CYL_FWD_I1100_2  ;
	1101: Lamp3:=I50_LH_REJ_CYL_FWD_I1101_2  ;
	1110: Lamp3:=I70_DRUM_FEED_CONV1_OVERFLW_I1110_2  ;
	1111: Lamp3:=I70_TOP_REJ_BIN_PRSNCE_I1111_2 ;
   ELSE
       Visibility_3:=FALSE;	
   END_CASE  
   
     CASE IP_Arr_OP10P[Input_Page_num] OF
     //300:  Line4:= "I10A_SPARE_I300_3(I300.3)              "  ;
     //301:  Line4:= "I10A_SPARE_I301_3(I301.3)              "  ;
     302:  Line4:= "I10B_DRUM_CONV_REV(I302.3)               "  ;
     303:  Line4:= "I10B_SPARE_I303_3(I303.3)                "  ;
     304:  Line4:= "I30_DRUM_CONV_REV(I304.3)                "  ;
     305:  Line4:= "I40_ATC_STN_POKE_YOKE_2(I305.3)          "  ;
     306:  Line4:= "I50_DRUM_CONV_REV(I306.3)                "  ;
     307:  Line4:= "I60_ATC_STN_POKE_YOKE_2(I307.3)          "  ;
     308:  Line4:= "I70_DRUM_CONV_REV(I308.3)                "  ;
     309:  Line4:= "I80_ATC_STN_POKE_YOKE_2(I309.3)          "  ;
     310:  Line4:= "I80_SPARE_I310_3(I310.3)                 "  ;
     311:  Line4:= "I80_SPARE_I311_3(I311.3)                 "  ;
     1000: Line4:= "I10A_SPARE_I1000_3(I1000.3)              "  ;
     1001: Line4:= "I10A_BDY1_PRSN_MOVER(I1001,3)            "  ;
     1010: Line4:= "I10A_ORING_LH_GRPR_OPN(I1010.3)          "  ;
     1011: Line4:= "I10A_ORING_HORZ_CYL_FWD(I1011.3)         "  ;
     1020: Line4:= "I10A_BDY_SING_CYL_OPN(I1020.3)           "  ;
     1021: Line4:= "I10A_SPARE_I1021_3(I1021.3)              "  ;
     1030: Line4:= "I10B_ORING_LH_GRPR_OPN(I1030.3)          "  ;
     1031: Line4:= "I10B_ORING_HORZ_CYL_FWD(I1031.3)         "  ;
     1040: Line4:= "I10B_BDY_SING_CYL_OPN(I1040.3)           "  ;
     1041: Line4:= "I10B_SPARE_I1041_3(I1041.3)              "  ;
     1100: Line4:= "I30_LH_REJ_CYL_REV(I1100.3)              "  ;
     1101: Line4:= "I50_LH_REJ_CYL_REV(I1101.3)              "  ;
     1110: Line4:= "I70_DRUM_FEED_CONV2_OVERFLW(I1110.3)     "  ;
     1111: Line4:= "I70_BOT_REJ_BIN_PRSNCE_I1111_3(I1111.3)  "  ;
     ELSE
     	Line4 := " ";
     END_CASE
	 
	 Visibility_4:=TRUE;
    CASE IP_Arr_OP10P[Input_Page_num] OF
	//300: Lamp4:=I10A_SPARE_I300_3;
	//301: Lamp4:=I10A_SPARE_I301_3;
	302: Lamp4:=I10B_DRUM_CONV_REV_I302_3 ;
	303: Lamp4:=I10B_SPARE_I303_3 ;
	304: Lamp4:=I30_DRUM_CONV_REV_I304_3;
	305: Lamp4:=I40_ATC_STN_POKE_YOKE_2_I305_3  ;
	306: Lamp4:=I50_DRUM_CONV_REV_I306_3;
	307: Lamp4:=I60_ATC_STN_POKE_YOKE_2_I307_3 ;
	308: Lamp4:=I70_DRUM_CONV_REV_I308_3 ;
	309: Lamp4:=I80_ATC_STN_POKE_YOKE_2_I309_3;
	310: Lamp4:=I80_SPARE_I310_3 ;
	311: Lamp4:=I80_SPARE_I311_3 ;
	1000: Lamp4:=I10A_SPARE_I1000_3  ;
	1001: Lamp4:=I10A_BDY1_PRSN_MOVER_I1001_3;
	1010: Lamp4:=I10A_ORING_LH_GRPR_OPN_I1010_3  ;
	1011: Lamp4:=I10A_ORING_HORZ_CYL_FWD_I1011_3  ;
	1020: Lamp4:=I10A_BDY_SING_CYL_OPN_I1020_3 ;
	1021: Lamp4:=I10A_SPARE_I1021_3 ;
	1030: Lamp4:=I10B_ORING_LH_GRPR_OPN_I1030_3 ;
	1031: Lamp4:=I10B_ORING_HORZ_CYL_FWD_I1031_3  ;
	1040: Lamp4:=I10B_BDY_SING_CYL_OPN_I1040_3  ;
	1041: Lamp4:=I10B_SPARE_I1041_3 ;
	1100: Lamp4:=I30_LH_REJ_CYL_REV_I1100_3 ;
	1101: Lamp4:=I50_LH_REJ_CYL_REV_I1101_3  ;
	1110: Lamp4:=I70_DRUM_FEED_CONV2_OVERFLW_I1110_3 ;
	1111: Lamp4:=I70_BOT_REJ_BIN_PRSNCE_I1111_3 ;
   ELSE
       Visibility_4:=FALSE;	
   END_CASE 
   
     CASE IP_Arr_OP10P[Input_Page_num] OF
     //300:  Line5:= "I10A_SPARE_I300_4(I300.4)             "  ;
     //301:  Line5:= "I10A_SPARE_I301_4(I301.4)             "  ;
     302:  Line5:= "I10B_DRUM_CONV_FWD(I302.4)              "  ;
     303:  Line5:= "I10B_SPARE_I303_4(I303.4)               "  ;
     304:  Line5:= "I30_DRUM_CONV_FWD(I304.4)               "  ;
     305:  Line5:= "I40_ATC_STN_POKE_YOKE_3(I305.4)         "  ;
     306:  Line5:= "I50_DRUM_CONV_FWD(I306.4)               "  ;
     307:  Line5:= "I60_ATC_STN_POKE_YOKE_3(I307.4)         "  ;
     308:  Line5:= "I70_DRUM_CONV_FWD(I308.4)               "  ;
     309:  Line5:= "I80_ATC_STN_POKE_YOKE_3(I309.4)         "  ;
     310:  Line5:= "I80_SPARE_I310_4(I310.4)                "  ;
     311:  Line5:= "I80_SPARE_I311_4(I311.4)                "  ;
     1000: Line5:= "I10A_SPARE_I1000_4(I1000.4)             "  ;
     1001: Line5:= "I10A_BDY2_PRSN_MOVER(I1001,4)           "  ;
     1010: Line5:= "I10A_ORING_LH_PUSHR_CYL_REV(I1010.4)    "  ;
     1011: Line5:= "I10A_ORING_VERT_CYL_UP(I1011.4)         "  ;
     1020: Line5:= "I10A_ORING_RH_GRPR_OPN(I1020.4)         "  ;
     1021: Line5:= "I10A_SPARE_I1021_4(I1021.4)             "  ;
     1030: Line5:= "I10B_ORING_LH_PUSHR_CYL_REV(I1030.4)    "  ;
     1031: Line5:= "I10B_ORING_VERT_CYL_UP(I1031.4)         "  ;
     1040: Line5:= "I10B_ORING_RH_GRPR_OPN(I1040.4)         "  ;
     1041: Line5:= "I10B_SPARE_I1041_4(I1041.4)             "  ;
     1100: Line5:= "I30_RH_REJ_CYL_FWD(I1100.4)             "  ;
     1101: Line5:= "I50_RH_REJ_CYL_FWD(I1101.4)             "  ;
     1110: Line5:= "I70_LH_REJ_CYL_FWD(I1110.4)             "  ;
     1111: Line5:= "I70_SPARE_I1111_4(I1111.4)		    "  ;
     ELSE
     	Line5 := " ";
     END_CASE
     
	 Visibility_5:=TRUE;	
	 CASE IP_Arr_OP10P[Input_Page_num] OF
	//300: Lamp5:=I10A_SPARE_I300_4;
	//301: Lamp5:=I10A_SPARE_I301_4;
	302: Lamp5:=I10B_DRUM_CONV_FWD_I302_4 ;
	303: Lamp5:=I10B_SPARE_I303_4 ;
	304: Lamp5:=I30_DRUM_CONV_FWD_I304_4 ;
	305: Lamp5:=I40_ATC_STN_POKE_YOKE_3_I305_4 ;
	306: Lamp5:=I50_DRUM_CONV_FWD_I306_4  ;
	307: Lamp5:=I60_ATC_STN_POKE_YOKE_3_I307_4  ;
	308: Lamp5:=I70_DRUM_CONV_FWD_I308_4 ;
	309: Lamp5:=I80_ATC_STN_POKE_YOKE_3_I309_4 ;
	310: Lamp5:=I80_SPARE_I310_4 ;
	311: Lamp5:=I80_SPARE_I311_4 ;
	1000:Lamp5:=I10A_SPARE_I1000_4 ;
	1001:Lamp5:=I10A_BDY2_PRSN_MOVER_I1001_4;
	1010:Lamp5:=I10A_ORING_LH_PUSHR_CYL_REV_I1010_4 ;
	1011:Lamp5:=I10A_ORING_VERT_CYL_UP_I1011_4   ;
	1020:Lamp5:=I10A_ORING_RH_GRPR_OPN_I1020_4;
	1021:Lamp5:=I10A_SPARE_I1021_4 ;
	1030:Lamp5:=I10B_ORING_LH_PUSHR_CYL_REV_I1030_4 ;
	1031:Lamp5:=I10B_ORING_VERT_CYL_UP_I1031_4  ;
	1040:Lamp5:=I10B_ORING_RH_GRPR_OPN_I1040_4 ;
	1041:Lamp5:=I10B_SPARE_I1041_4;
	1100:Lamp5:=I30_RH_REJ_CYL_FWD_I1100_4  ;
	1101:Lamp5:=I50_RH_REJ_CYL_FWD_I1101_4 ;
	1110:Lamp5:=I70_LH_REJ_CYL_FWD_I1110_4;
	1111:Lamp5:=I70_SPARE_I1111_4 ;
   ELSE
       Visibility_5:=FALSE;	
   END_CASE
	 
     CASE IP_Arr_OP10P[Input_Page_num] OF
     //300:  Line6:= "I10A_SPARE_I300_5(I300.5)          "  ;
     //301:  Line6:= "I10A_SPARE_I301_5(I301.5)          "  ;
     302:  Line6:= "I10B_ROB_MAN_AUTO_MODE(I302.5)       "  ;
     303:  Line6:= "I10B_SPARE_I303_5(I303.5)            "  ;
     304:  Line6:= "I30_SPARE_I304_5(I304.5)             "  ;
     305:  Line6:= "I40_ATC_STN_POKE_YOKE_4(I305.5)      "  ;
     306:  Line6:= "I50_SPARE_I306_5(I306.5)             "  ;
     307:  Line6:= "I60_ATC_STN_POKE_YOKE_4(I307.5)      "  ;
     308:  Line6:= "I70_SPARE_I308_5(I308.5)             "  ;
     309:  Line6:= "I80_ATC_STN_POKE_YOKE_4(I309.5)      "  ;
     310:  Line6:= "I80_SPARE_I310_5(I310.5)             "  ;
     311:  Line6:= "I80_SPARE_I311_5(I311.5)             "  ;
     1000: Line6:= "I10_LH_LNR_TRK_BDY_PRSN(I1000.5)     "  ;
     1001: Line6:= "I10B_BDY1_PRSN_MOVER(I1001,5)        "  ;
     1010: Line6:= "I10A_ORING_RH_GRPR_OPN_I1010_5(I1010.5) "  ;
     1011: Line6:= "I10A_ORING_VERT_CYL_DWN(I1011.5)     "  ;
     1020: Line6:= "I10A_ORING_RH_PUSHR_CYL_FWD(I1020.5) "  ;
     1021: Line6:= "I10A_SPARE_I1021_5(I1021.5)          "  ;
     1030: Line6:= "I10B_ORING_RH_GRPR_OPN_I1030_5(I1030.5) "  ;
     1031: Line6:= "I10B_ORING_VERT_CYL_DWN(I1031.5)     "  ;
     1040: Line6:= "I10B_ORING_RH_PUSHR_CYL_FWD(I1040.5  "  ;
     1041: Line6:= "I10B_SPARE_I1041_5(I1041.5)          "  ;
     1100: Line6:= "I30_RH_REJ_CYL_REV(I1100.5)          "  ;
     1101: Line6:= "I50_RH_REJ_CYL_REV(I1101.5)          "  ;
     1110: Line6:= "I70_LH_REJ_CYL_REV(I1110.5)          "  ;
     1111: Line6:= "I70_SPARE_I1111.5(I1111.5)           "  ;
     ELSE
     	Line6 := " ";
     END_CASE
     Visibility_6:=TRUE;
	CASE IP_Arr_OP10P[Input_Page_num] OF
	//300: Lamp6:=I10A_SPARE_I300_5 ;
	//301: Lamp6:=I10A_SPARE_I301_5;
	302: Lamp6:=I10B_ROB_MAN_AUTO_MODE_I302_5 ;
	303: Lamp6:=I10B_SPARE_I303_5 ;
	304: Lamp6:=I30_SPARE_I304_5;
	305: Lamp6:=I40_ATC_STN_POKE_YOKE_4_I305_5  ;
	306: Lamp6:=I50_SPARE_I306_5;
	307: Lamp6:=I60_ATC_STN_POKE_YOKE_4_I307_5 ;
	308: Lamp6:=I70_SPARE_I308_5 ;
	309: Lamp6:=I80_ATC_STN_POKE_YOKE_4_I309_5;
	310: Lamp6:=I80_SPARE_I310_5;
	311: Lamp6:=I80_SPARE_I311_5;
	1000: Lamp6:=I10_LH_LNR_TRK_BDY_PRSN_I1000_5  ;
	1001: Lamp6:=I10B_BDY1_PRSN_MOVER_I1001_5;
	1010: Lamp6:=I10A_ORING_RH_GRPR_OPN_I1010_5 ;
	1011: Lamp6:=I10A_ORING_VERT_CYL_DWN_I1011_5  ;
	1020: Lamp6:=I10A_ORING_RH_PUSHR_CYL_FWD_I1020_5 ;
	1021: Lamp6:=I10A_SPARE_I1021_5 ;
	1030: Lamp6:=I10B_ORING_RH_GRPR_OPN_I1030_5 ;
	1031: Lamp6:=I10B_ORING_VERT_CYL_DWN_I1031_5   ;
	1040: Lamp6:=I10B_ORING_RH_PUSHR_CYL_FWD_I1040_5  ;
	1041: Lamp6:=I10B_SPARE_I1041_5 ;
	1100: Lamp6:=I30_RH_REJ_CYL_REV_I1100_5 ;
	1101: Lamp6:=I50_RH_REJ_CYL_REV_I1101_5  ;
	1110: Lamp6:=I70_LH_REJ_CYL_REV_I1110_5  ;
	1111: Lamp6:=I70_SPARE_I1111_5  ;
   ELSE
       Visibility_6:=FALSE;	
   END_CASE
	 
     CASE IP_Arr_OP10P[Input_Page_num] OF
     //300:  Line7:= "I10A_SPARE_I300_6(I300.6)     "  ;
     //301:  Line7:= "I10A_SPARE_I301_6(I301.6)     "  ;
     302:  Line7:= "I10B_SPARE_I302_6(I302.6)       "  ;
     303:  Line7:= "I10B_SPARE_I303_6(I303.6)       "  ;
     304:  Line7:= "I30_SPARE_I304_6(I304.6)        "  ;
     305:  Line7:= "I40_ATC_SLAVE_MODL1(I305.6)     "  ;
     306:  Line7:= "I50_SPARE_I306_6(I306.6)        "  ;
     307:  Line7:= "I60_ATC_SLAVE_MODL1(I307.6)     "  ;
     308:  Line7:= "I70_SPARE_I308_6(I308.6)        "  ;
     309:  Line7:= "I80_ATC_SLAVE_MODL1(I309.6)     "  ;
     310:  Line7:= "I80_SPARE_I310_6(I310.6)        "  ;
     311:  Line7:= "I80_SPARE_I311_6(I311.6)        "  ;
     1000: Line7:= "I10_RH_LNR_TRK_BDY_PRSN(I1000.6)"  ;
     1001: Line7:= "I10B_BDY2_PRSN_MOVER(I1001,6)   "  ;
     1010: Line7:= "I10A_ORING_RH_GRPR_CLSE(I1010.6)"  ;
     1011: Line7:= "I10A_LH_FIRTRE_ORING_REJ_CYL_REV(I1011.6) "  ;
     1020: Line7:= "I10A_ORING_REJ_BIN_PRSNCE(I1020.6)     "  ;
     1021: Line7:= "I10A_SPARE_I1021_6(I1021.6)     "  ;
     1030: Line7:= "I10B_ORING_RH_GRPR_CLSE(I1030.6)"  ;
     1031: Line7:= "I10B_LH_FIRTRE_ORING_REJ_CYL_REV(I1031.6) "  ;
     1040: Line7:= "I10B_ORING_REJ_BIN_PRSNCE_I1040_6(I1040.6)"  ;
     1041: Line7:= "I10B_SPARE_I1041_6(I1041.6)     "  ;
     1100: Line7:= "I30_TOP_REJ_BIN_PRSNCE_I1100_6(I1100.6)"  ;
     1101: Line7:= "I50_SPARE_I1101_6(I1101.6)        "  ;
     1110: Line7:= "I70_RH_REJ_CYL_FWD(I1110.6)     "  ;
     1111: Line7:= "I70_SPARE_I1111_6(I1111.6)	   "  ;
     ELSE
     	Line7 := " ";
     END_CASE
     Visibility_7:=TRUE;
	 CASE IP_Arr_OP10P[Input_Page_num] OF
	//300: Lamp7:=I10A_SPARE_I300_6 ;
	//301: Lamp7:=I10A_SPARE_I301_6;
	302: Lamp7:=I10B_SPARE_I302_6 ;
	303: Lamp7:=I10B_SPARE_I303_6 ;
	304: Lamp7:=I30_SPARE_I304_6 ;
	305: Lamp7:=I40_ATC_SLAVE_MODL1_I305_6   ;
	306: Lamp7:=I50_SPARE_I306_6 ;
	307: Lamp7:=I60_ATC_SLAVE_MODL1_I307_6 ;
	308: Lamp7:=I70_SPARE_I308_6 ;
	309: Lamp7:=I80_ATC_SLAVE_MODL1_I309_6 ;
	310: Lamp7:=I80_SPARE_I310_6;
	311: Lamp7:=I80_SPARE_I311_6;
	1000:Lamp7:=I10_RH_LNR_TRK_BDY_PRSN_I1000_6 ;
	1001:Lamp7:=I10B_BDY2_PRSN_MOVER_I1001_6;
	1010:Lamp7:=I10A_ORING_RH_GRPR_CLSE_I1010_6 ;
	1011:Lamp7:=I10A_LH_FIRTRE_ORING_REJ_CYL_REV_I1011_6   ;
	1020:Lamp7:=I10A_ORING_REJ_BIN_PRSNCE_I1020_6;
	1021:Lamp7:=I10A_SPARE_I1021_6 ;
	1030:Lamp7:=I10B_ORING_RH_GRPR_CLSE_I1030_6 ;
	1031:Lamp7:=I10B_LH_FIRTRE_ORING_REJ_CYL_REV_I1031_6 ;
	1040:Lamp7:=I10B_ORING_REJ_BIN_PRSNCE_I1040_6 ;
	1041:Lamp7:=I10B_SPARE_I1041_6;
	1100:Lamp7:=I30_TOP_REJ_BIN_PRSNCE_I1100_6 ;
	1101:Lamp7:=I50_SPARE_I1101_6 ;
	1110:Lamp7:=I70_RH_REJ_CYL_FWD_I1110_6   ;
	1111:Lamp7:=I70_SPARE_I1111_6   ;
   ELSE
       Visibility_7:=FALSE;	
   END_CASE 
	 
     CASE IP_Arr_OP10P[Input_Page_num] OF
     //300:  Line8:= "I10A_SPARE_I300_7(I300.7)       "  ;
     //301:  Line8:= "I10A_SPARE_I301_7(I301.7)       "  ;
     302:  Line8:= "I10B_SPARE_I302_7(I302.7)       "  ;
     303:  Line8:= "I10B_SPARE_I303_7(I303.7)       "  ;
     304:  Line8:= "I30_SPARE_I304_7(I304.7)        "  ;
     305:  Line8:= "I40_ATC_SLAVE_MODL2(I305.7)     "  ;
     306:  Line8:= "I50_SPARE_I306_7(I306.7)        "  ;
     307:  Line8:= "I60_ATC_SLAVE_MODL2(I307.7)     "  ;
     308:  Line8:= "I70_SPARE_I308_7(I308.7)        "  ;
     309:  Line8:= "I80_ATC_SLAVE_MODL2(I309.7)     "  ;
     310:  Line8:= "I80_SPARE_I310_7(I310.7)        "  ;
     311:  Line8:= "I80_SPARE_I311_7(I311.7)        "  ;
     1000: Line8:= "I10_LH_LNR_TRCK_FIX_CHO_1_I1000_7(I1000.7)     "  ;
     1001: Line8:= "I10B_SPARE_I1001_7(I1001,7)     "  ;
     1010: Line8:= "I10A_ORING_RH_PUSHR_CYL_REV(I1010.7) "  ;
     1011: Line8:= "I10A_LH_FIRTRE_ORING_REJ_CYL_FWD(I1011.7)"  ;
     1020: Line8:= "I10A_BOWL_TRK_INDXR_POS1(I1020.7)     "  ;
     1021: Line8:= "I10A_SPARE_I1021_7(I1021.7)     "  ;
     1030: Line8:= "I10B_ORING_RH_PUSHR_CYL_REV(I1030.7)"  ;
     1031: Line8:= "I10B_LH_FIRTRE_ORING_REJ_CYL_FWD(I1031.7)"  ;
     1040: Line8:= "I10B_BOWL_TRK_INDXR_POS1(I1040.7)     "  ;
     1041: Line8:= "I10B_SPARE_I1041_7(I1041.7)     "  ;
     1100: Line8:= "I30_BOT_REJ_BIN_PRSNCE(I1100.7)      "  ;
     1101: Line8:= "O50_LH_GRIP_CLSE(I1101.7)       "  ;
     1110: Line8:= "I70_RH_REJ_CYL_REV(I1110.7)     "  ;
     1111: Line8:= "I70_SPARE_I1111_7(I1111.7)      "  ;
     ELSE
     	Line8 := " ";
     END_CASE
     
	Visibility_8:=TRUE;	 
    CASE IP_Arr_OP10P[Input_Page_num] OF
	//300: Lamp8:=I10A_SPARE_I300_7 ;
	//301: Lamp8:=I10A_SPARE_I301_7;
	302: Lamp8:=I10B_SPARE_I302_7 ;
	303: Lamp8:=I10B_SPARE_I303_7;
	304: Lamp8:=I30_SPARE_I304_7 ;
	305: Lamp8:=I40_ATC_SLAVE_MODL2_I305_7  ;
	306: Lamp8:=I50_SPARE_I306_7 ;
	307: Lamp8:=I60_ATC_SLAVE_MODL2_I307_7 ;
	308: Lamp8:=I70_SPARE_I308_7 ;
	309: Lamp8:=I80_ATC_SLAVE_MODL2_I309_7 ;
	310: Lamp8:=I80_SPARE_I310_7;
	311: Lamp8:=I80_SPARE_I311_7 ;
	1000:Lamp8:=I10_LH_LNR_TRCK_FIX_CHO_1_I1000_7   ;
	1001:Lamp8:=I10A_SPARE_I1001_7 ;
	1010:Lamp8:=I10A_ORING_RH_PUSHR_CYL_REV_I1010_7   ;
	1011:Lamp8:=I10A_LH_FIRTRE_ORING_REJ_CYL_FWD_I1011_7    ;
	1020:Lamp8:=I10A_BOWL_TRK_INDXR_POS1_I1020_7 ;
	1021:Lamp8:=I10A_SPARE_I1021_7  ;
	1030:Lamp8:=I10B_ORING_RH_PUSHR_CYL_REV_I1030_7;
	1031:Lamp8:=I10B_LH_FIRTRE_ORING_REJ_CYL_FWD_I1031_7;
	1040:Lamp8:=I10B_BOWL_TRK_INDXR_POS1_I1040_7 ;
	1041:Lamp8:=I10B_SPARE_I1041_7 ;
	1100:Lamp8:=I30_BOT_REJ_BIN_PRSNCE_I1100_7;
	1101:Lamp8:=I50_LH_GRIP_CLSE_I1101_7 ;
	1110:Lamp8:=I70_RH_REJ_CYL_REV_I1110_7  ;
	1111:Lamp8:=I70_SPARE_I1111_7 ;
   ELSE
       Visibility_8:=FALSE;	
   END_CASE 
     
     CASE OP_Arr_OP10P[Output_Page_num] OF
     300: OLine1:= "O10_XTS_GREASE_VALVE_ON(Q300.0)  ";
     301: OLine1:= "O10A_BDY_EMPT_CAM_LGHT1_ON(Q301.0)     ";
     302: OLine1:= "O10B_DRUM_MTR_FWD(Q302.0)              ";
     303: OLine1:= "O10_TWR_LMP_BUZZ(Q303.0)             ";
     304: OLine1:= "O20_SPARE_Q304_0(Q304.0)             ";
     305: OLine1:= "O30_DRUM_RUN_IND(Q305.0)             ";
     306: OLine1:= "O50_DRUM_EXT_SPEED(Q306.0)              ";
     307: OLine1:= "O50_BARLIGHT_OP2(Q307.0)             ";
     308: OLine1:= "O70_BARLIGHT_OP1(Q308.0)              ";
     309: OLine1:= "O70_SPARE_Q309_0(Q309.0)              ";
     1050: OLine1:= "O10A_ORING_LH_GRPR_CLSE_OPN(Q1050.0) ";
     1051: OLine1:= "O10A_ORING_VERT_CYL_UP(Q1051.0)     ";
     1052: OLine1:= "O10A_SPARE_Q1052_0(Q1052.0)         ";
     1053: OLine1:= "O10A_SPARE_Q1053_0(Q1053.0)         ";
     1060: OLine1:= "O10B_ORING_LH_GRPR_CLSE_OPN(Q1060.0) ";
     1061: OLine1:= "O10B_ORING_VERT_CYL_UP(Q1061.0)     ";
     1062: OLine1:= "O10B_DRUM_FEED_AIRPURGE_ON(Q1062.0) ";
     1063: OLine1:= "O10B_SPARE_Q1063_0(Q1063.0)        ";
     1150: OLine1:= "O20_LH_OIL_DISPN_ON(Q1150.0)         ";
     1151: OLine1:= "O40_TOOL_CHO_UNLOCK(Q1151.0)         ";
     1152: OLine1:= "O50_RH_REJ_CYL_FWD_REV(Q1152.0)     ";
     1153: OLine1:= "O80_TOOL_CHO_UNLOCK(Q1153.0)			";	
     ELSE
     	OLine1 := " ";
     END_CASE
      Out_Visibility_1:=TRUE;
   
   CASE OP_Arr_OP10P[Output_Page_num] OF
	300:  Out_Lamp1:=O10_XTS_GREASE_VALVE_ON_Q300_0;
	301:  Out_Lamp1:=O10A_BDY_EMPT_CAM_LGHT1_ON_Q301_0;
	302:  Out_Lamp1:=O10B_DRUM_MTR_FWD_Q302_0;
	303:  Out_Lamp1:=O10_TWR_LMP_BUZZ_Q303_0;
	304:  Out_Lamp1:=O20_SPARE_Q304_0;
	305:  Out_Lamp1:=O30_DRUM_RUN_IND_Q305_0;
	306:  Out_Lamp1:=O50_DRUM_EXT_SPEED_Q306_0;
	307:  Out_Lamp1:=O50_BARLIGHT_OP2_Q307_0;
	308:  Out_Lamp1:=O70_BARLIGHT_OP1_Q308_0;
	309:  Out_Lamp1:=O70_SPARE_Q309_0;
	1050: Out_Lamp1:=O10A_ORING_LH_GRPR_CLSE_OPN_Q1050_0;
	1051: Out_Lamp1:=O10A_ORING_VERT_CYL_UP_Q1051_0;
	1052: Out_Lamp1:=O10A_SPARE_Q1052_0;
	1053: Out_Lamp1:=O10A_SPARE_Q1053_0;
	1060: Out_Lamp1:=O10B_ORING_LH_GRPR_CLSE_OPN_Q1060_0;
	1061: Out_Lamp1:=O10B_ORING_VERT_CYL_UP_Q1061_0;
	1062: Out_Lamp1:=O10B_DRUM_FEED_AIRPURGE_ON_Q1062_0;
	1063: Out_Lamp1:=O10B_SPARE_Q1063_0;
	1150: Out_Lamp1:=O20_LH_OIL_DISPN_ON_Q1150_0;
	1151: Out_Lamp1:=O40_TOOL_CHO_UNLOCK_Q1151_0;
	1152: Out_Lamp1:=O50_RH_REJ_CYL_REV_Q1152_0;
	1153: Out_Lamp1:=O80_TOOL_CHO_UNLOCK_Q1153_0;
   ELSE
       Out_Visibility_1:=FALSE;	
   END_CASE
   
